  MoveL 11373 to (499.02, 502.81, 19.8) mm, rotated rx 0 ry 90 rz 0 deg; joints [-12.285, -28.387, 111.814, -16.313, -82.826, 51.071]
  Set speed (15.0 mm/s)
  Call Extruder(0.024)
  MoveL 11374 to (498.43, 503.4, 19.8) mm, rotated rx 0 ry 90 rz 0 deg; joints [-12.351, -28.396, 111.869, -16.378, -82.873, 51.065]
  Set speed (120.0 mm/s)
  MoveL 11375 to (496.44, 504.19, 19.8) mm, rotated rx 0 ry 90 rz 0 deg; joints [-12.464, -28.43, 112.084, -16.485, -83.05, 51.026]
  Set speed (1000.0 mm/s)
  MoveL 11376 to (495, 504.85, 19.8) mm, rotated rx 0 ry 90 rz 0 deg; joints [-12.554, -28.454, 112.239, -16.571, -83.178, 50.998]
  Set speed (15.0 mm/s)
  Call Extruder(0.148)
  MoveL 11377 to (491.4, 508.44, 19.8) mm, rotated rx 0 ry 90 rz 0 deg; joints [-12.96, -28.505, 112.569, -16.971, -83.458, 50.958]
  Set speed (120.0 mm/s)
  MoveL 11378 to (492.24, 508.59, 19.8) mm, rotated rx 0 ry 90 rz 0 deg; joints [-12.956, -28.489, 112.465, -16.97, -83.374, 50.983]
  Set speed (15.0 mm/s)
  Call Extruder(0.113)
  MoveL 11379 to (495, 505.84, 19.8) mm, rotated rx 0 ry 90 rz 0 deg; joints [-12.645, -28.45, 112.212, -16.664, -83.16, 51.014]
  Set speed (120.0 mm/s)
  MoveL 11380 to (495, 506.83, 19.8) mm, rotated rx 0 ry 90 rz 0 deg; joints [-12.735, -28.446, 112.186, -16.756, -83.141, 51.03]
  Set speed (15.0 mm/s)
  Call Extruder(0.073)
  MoveL 11381 to (493.23, 508.59, 19.8) mm, rotated rx 0 ry 90 rz 0 deg; joints [-12.935, -28.471, 112.348, -16.952, -83.278, 51.01]
  Set speed (120.0 mm/s)
  MoveL 11382 to (494.22, 508.59, 19.8) mm, rotated rx 0 ry 90 rz 0 deg; joints [-12.914, -28.453, 112.23, -16.934, -83.183, 51.037]
  Set speed (15.0 mm/s)
  Call Extruder(0.036)
  MoveL 11383 to (495.1, 507.72, 19.8) mm, rotated rx 0 ry 90 rz 0 deg; joints [-12.816, -28.441, 112.15, -16.838, -83.115, 51.047]
  Set speed (120.0 mm/s)
  MoveL 11384 to (495.21, 508.59, 19.8) mm, rotated rx 0 ry 90 rz 0 deg; joints [-12.893, -28.435, 112.113, -16.917, -83.087, 51.064]
  Set speed (15.0 mm/s)
  MoveL 11385 to (496.09, 507.72, 19.8) mm, rotated rx 0 ry 90 rz 0 deg; joints [-12.795, -28.422, 112.033, -16.82, -83.019, 51.074]
  Set speed (120.0 mm/s)
  MoveL 11386 to (496.2, 508.59, 19.8) mm, rotated rx 0 ry 90 rz 0 deg; joints [-12.872, -28.416, 111.995, -16.899, -82.992, 51.091]
  Set speed (15.0 mm/s)
  Call Extruder(0.036)
  MoveL 11387 to (497.08, 507.72, 19.8) mm, rotated rx 0 ry 90 rz 0 deg; joints [-12.774, -28.403, 111.915, -16.803, -82.924, 51.1]
  Set speed (120.0 mm/s)
  MoveL 11388 to (497.19, 508.59, 19.8) mm, rotated rx 0 ry 90 rz 0 deg; joints [-12.852, -28.397, 111.877, -16.882, -82.896, 51.118]
  Set speed (15.0 mm/s)
  MoveL 11389 to (498.07, 507.72, 19.8) mm, rotated rx 0 ry 90 rz 0 deg; joints [-12.754, -28.385, 111.797, -16.786, -82.828, 51.127]
  Set speed (120.0 mm/s)
  MoveL 11390 to (498.18, 508.59, 19.8) mm, rotated rx 0 ry 90 rz 0 deg; joints [-12.831, -28.379, 111.759, -16.865, -82.801, 51.145]
  Set speed (15.0 mm/s)
  MoveL 11391 to (499.06, 507.72, 19.8) mm, rotated rx 0 ry 90 rz 0 deg; joints [-12.733, -28.366, 111.679, -16.769, -82.733, 51.153]
  Set speed (120.0 mm/s)
  MoveL 11392 to (499.17, 508.59, 19.8) mm, rotated rx 0 ry 90 rz 0 deg; joints [-12.811, -28.36, 111.641, -16.848, -82.705, 51.171]
  Set speed (15.0 mm/s)
  MoveL 11393 to (500.05, 507.72, 19.8) mm, rotated rx 0 ry 90 rz 0 deg; joints [-12.713, -28.347, 111.561, -16.752, -82.637, 51.18]
  Set speed (120.0 mm/s)
  MoveL 11394 to (500.16, 508.59, 19.8) mm, rotated rx 0 ry 90 rz 0 deg; joints [-12.79, -28.34, 111.523, -16.831, -82.61, 51.198]
  Set speed (15.0 mm/s)
  MoveL 11395 to (501.04, 507.72, 19.8) mm, rotated rx 0 ry 90 rz 0 deg; joints [-12.693, -28.327, 111.443, -16.735, -82.542, 51.206]
  Set speed (120.0 mm/s)
  MoveL 11396 to (501.15, 508.59, 19.8) mm, rotated rx 0 ry 90 rz 0 deg; joints [-12.77, -28.321, 111.405, -16.814, -82.514, 51.224]
  Set speed (15.0 mm/s)
  MoveL 11397 to (502.03, 507.72, 19.8) mm, rotated rx 0 ry 90 rz 0 deg; joints [-12.672, -28.308, 111.324, -16.719, -82.446, 51.233]
  Set speed (120.0 mm/s)
  MoveL 11398 to (502.14, 508.59, 19.8) mm, rotated rx 0 ry 90 rz 0 deg; joints [-12.749, -28.302, 111.287, -16.797, -82.419, 51.251]
  Set speed (15.0 mm/s)
  MoveL 11399 to (503.02, 507.72, 19.8) mm, rotated rx 0 ry 90 rz 0 deg; joints [-12.652, -28.288, 111.206, -16.702, -82.351, 51.259]
  Set speed (120.0 mm/s)
  MoveL 11400 to (503.13, 508.59, 19.8) mm, rotated rx 0 ry 90 rz 0 deg; joints [-12.729, -28.282, 111.168, -16.781, -82.324, 51.277]
  Set speed (15.0 mm/s)
  MoveL 11401 to (504.01, 507.72, 19.8) mm, rotated rx 0 ry 90 rz 0 deg; joints [-12.632, -28.268, 111.087, -16.686, -82.255, 51.285]
  Set speed (120.0 mm/s)
  MoveL 11402 to (504.12, 508.59, 19.8) mm, rotated rx 0 ry 90 rz 0 deg; joints [-12.709, -28.262, 111.049, -16.764, -82.228, 51.304]
  Set speed (15.0 mm/s)
  MoveL 11403 to (505, 507.72, 19.8) mm, rotated rx 0 ry 90 rz 0 deg; joints [-12.612, -28.249, 110.968, -16.669, -82.16, 51.311]
  Set speed (120.0 mm/s)
  MoveL 11404 to (505.33, 507.39, 19.8) mm, rotated rx 0 ry 90 rz 0 deg; joints [-12.575, -28.243, 110.937, -16.633, -82.134, 51.314]
  Set speed (15.0 mm/s)
  Call Extruder(0.134)
  MoveL 11405 to (508.59, 504.12, 19.8) mm, rotated rx 0 ry 90 rz 0 deg; joints [-12.216, -28.191, 110.631, -16.281, -81.877, 51.342]
  Set speed (120.0 mm/s)
  MoveL 11406 to (508.59, 505.11, 19.8) mm, rotated rx 0 ry 90 rz 0 deg; joints [-12.305, -28.187, 110.605, -16.371, -81.86, 51.36]
  Set speed (15.0 mm/s)
  Call Extruder(0.143)
  MoveL 11407 to (505.11, 508.59, 19.8) mm, rotated rx 0 ry 90 rz 0 deg; joints [-12.689, -28.242, 110.931, -16.748, -82.133, 51.33]
  Set speed (120.0 mm/s)
  MoveL 11408 to (506.1, 508.59, 19.8) mm, rotated rx 0 ry 90 rz 0 deg; joints [-12.668, -28.222, 110.812, -16.732, -82.038, 51.356]
  Set speed (15.0 mm/s)
  Call Extruder(0.103)
  MoveL 11409 to (508.59, 506.1, 19.8) mm, rotated rx 0 ry 90 rz 0 deg; joints [-12.394, -28.182, 110.579, -16.462, -81.842, 51.377]
  Set speed (120.0 mm/s)
  MoveL 11410 to (508.59, 507.09, 19.8) mm, rotated rx 0 ry 90 rz 0 deg; joints [-12.483, -28.178, 110.552, -16.553, -81.825, 51.395]
  Set speed (15.0 mm/s)
  Call Extruder(0.062)
  MoveL 11411 to (507.09, 508.59, 19.8) mm, rotated rx 0 ry 90 rz 0 deg; joints [-12.648, -28.202, 110.693, -16.715, -81.942, 51.382]
  Set speed (120.0 mm/s)
  MoveL 11412 to (508.08, 508.59, 19.8) mm, rotated rx 0 ry 90 rz 0 deg; joints [-12.628, -28.181, 110.574, -16.699, -81.847, 51.408]
  Set speed (15.0 mm/s)
  Call Extruder(0.021)
  MoveL 11413 to (508.59, 508.08, 19.8) mm, rotated rx 0 ry 90 rz 0 deg; joints [-12.572, -28.173, 110.526, -16.644, -81.807, 51.413]
  Set speed (120.0 mm/s)
  MoveL 11414 to (505.33, 506.39, 19.8) mm, rotated rx 0 ry 90 rz 0 deg; joints [-12.485, -28.248, 110.963, -16.542, -82.152, 51.297]
  Set speed (15.0 mm/s)
  Call Extruder(0.134)
  MoveL 11415 to (508.59, 503.13, 19.8) mm, rotated rx 0 ry 90 rz 0 deg; joints [-12.126, -28.195, 110.656, -16.19, -81.894, 51.325]
  Set speed (120.0 mm/s)
  MoveL 11416 to (508.59, 502.14, 19.8) mm, rotated rx 0 ry 90 rz 0 deg; joints [-12.037, -28.2, 110.682, -16.099, -81.911, 51.307]
  Set speed (15.0 mm/s)
  Call Extruder(0.136)
  MoveL 11417 to (505.28, 505.46, 19.8) mm, rotated rx 0 ry 90 rz 0 deg; joints [-12.402, -28.253, 110.994, -16.456, -82.173, 51.279]
  Set speed (120.0 mm/s)
  MoveL 11418 to (504.94, 504.8, 19.8) mm, rotated rx 0 ry 90 rz 0 deg; joints [-12.349, -28.263, 111.052, -16.401, -82.217, 51.259]
  Set speed (15.0 mm/s)
  Call Extruder(0.150)
  MoveL 11419 to (508.59, 501.15, 19.8) mm, rotated rx 0 ry 90 rz 0 deg; joints [-11.948, -28.204, 110.707, -16.008, -81.928, 51.29]
  Set speed (120.0 mm/s)
  MoveL 11420 to (508.59, 500.16, 19.8) mm, rotated rx 0 ry 90 rz 0 deg; joints [-11.858, -28.208, 110.732, -15.916, -81.945, 51.273]
  Set speed (15.0 mm/s)
  Call Extruder(0.164)
  MoveL 11421 to (504.61, 504.15, 19.8) mm, rotated rx 0 ry 90 rz 0 deg; joints [-12.296, -28.272, 111.109, -16.346, -82.261, 51.239]
  Set speed (120.0 mm/s)
  MoveL 11422 to (504.27, 503.49, 19.8) mm, rotated rx 0 ry 90 rz 0 deg; joints [-12.243, -28.282, 111.167, -16.291, -82.305, 51.219]
  Set speed (15.0 mm/s)
  Call Extruder(0.178)
  MoveL 11423 to (508.59, 499.17, 19.8) mm, rotated rx 0 ry 90 rz 0 deg; joints [-11.769, -28.213, 110.757, -15.825, -81.962, 51.256]
  Set speed (120.0 mm/s)
  MoveL 11424 to (508.59, 498.18, 19.8) mm, rotated rx 0 ry 90 rz 0 deg; joints [-11.679, -28.217, 110.782, -15.734, -81.978, 51.239]
  Set speed (15.0 mm/s)
  Call Extruder(0.192)
  MoveL 11425 to (503.94, 502.84, 19.8) mm, rotated rx 0 ry 90 rz 0 deg; joints [-12.191, -28.291, 111.224, -16.236, -82.349, 51.2]
  Set speed (120.0 mm/s)
  MoveL 11426 to (503.6, 502.18, 19.8) mm, rotated rx 0 ry 90 rz 0 deg; joints [-12.138, -28.301, 111.281, -16.181, -82.393, 51.18]
  Set speed (15.0 mm/s)
  Call Extruder(0.205)
  MoveL 11427 to (508.59, 497.19, 19.8) mm, rotated rx 0 ry 90 rz 0 deg; joints [-11.589, -28.221, 110.807, -15.643, -81.995, 51.222]
  Set speed (120.0 mm/s)
  MoveL 11428 to (508.59, 496.2, 19.8) mm, rotated rx 0 ry 90 rz 0 deg; joints [-11.5, -28.225, 110.831, -15.552, -82.011, 51.206]
  Set speed (15.0 mm/s)
  Call Extruder(0.219)
  MoveL 11429 to (503.27, 501.53, 19.8) mm, rotated rx 0 ry 90 rz 0 deg; joints [-12.084, -28.31, 111.338, -16.126, -82.437, 51.16]
  Set speed (120.0 mm/s)
  MoveL 11430 to (502.93, 500.87, 19.8) mm, rotated rx 0 ry 90 rz 0 deg; joints [-12.031, -28.32, 111.395, -16.07, -82.481, 51.141]
  Set speed (15.0 mm/s)
  Call Extruder(0.233)
  MoveL 11431 to (508.59, 495.21, 19.8) mm, rotated rx 0 ry 90 rz 0 deg; joints [-11.41, -28.229, 110.855, -15.46, -82.028, 51.189]
  Set speed (120.0 mm/s)
  MoveL 11432 to (508.59, 494.22, 19.8) mm, rotated rx 0 ry 90 rz 0 deg; joints [-11.32, -28.234, 110.879, -15.369, -82.044, 51.172]
  Set speed (15.0 mm/s)
  Call Extruder(0.247)
  MoveL 11433 to (502.6, 500.22, 19.8) mm, rotated rx 0 ry 90 rz 0 deg; joints [-11.978, -28.329, 111.452, -16.015, -82.525, 51.121]
  Set speed (120.0 mm/s)
  MoveL 11434 to (502.26, 499.57, 19.8) mm, rotated rx 0 ry 90 rz 0 deg; joints [-11.925, -28.338, 111.509, -15.96, -82.569, 51.102]
  Set speed (15.0 mm/s)
  Call Extruder(0.109)
  MoveL 11435 to (504.9, 496.92, 19.8) mm, rotated rx 0 ry 90 rz 0 deg; joints [-11.634, -28.297, 111.258, -15.674, -82.358, 51.125]
  Set speed (120.0 mm/s)
  MoveL 11436 to (505.52, 496.31, 19.8) mm, rotated rx 0 ry 90 rz 0 deg; joints [-11.567, -28.287, 111.199, -15.608, -82.309, 51.131]
  Set speed (15.0 mm/s)
  Call Extruder(0.127)
  MoveL 11437 to (508.59, 493.23, 19.8) mm, rotated rx 0 ry 90 rz 0 deg; joints [-11.23, -28.238, 110.903, -15.277, -82.06, 51.156]
  Set speed (120.0 mm/s)
  MoveL 11438 to (508.59, 492.24, 19.8) mm, rotated rx 0 ry 90 rz 0 deg; joints [-11.14, -28.242, 110.927, -15.186, -82.076, 51.139]
  Set speed (15.0 mm/s)
  MoveL 11439 to (505.52, 495.32, 19.8) mm, rotated rx 0 ry 90 rz 0 deg; joints [-11.476, -28.291, 111.224, -15.516, -82.325, 51.114]
  Set speed (120.0 mm/s)
  MoveL 11440 to (505.52, 494.33, 19.8) mm, rotated rx 0 ry 90 rz 0 deg; joints [-11.386, -28.295, 111.248, -15.424, -82.342, 51.098]
  Set speed (15.0 mm/s)
  Call Extruder(0.121)
  MoveL 11441 to (508.44, 491.4, 19.8) mm, rotated rx 0 ry 90 rz 0 deg; joints [-11.067, -28.248, 110.965, -15.11, -82.104, 51.122]
  Set speed (120.0 mm/s)
  MoveL 11442 to (507.45, 491.4, 19.8) mm, rotated rx 0 ry 90 rz 0 deg; joints [-11.084, -28.268, 111.084, -15.125, -82.2, 51.098]
  Set speed (15.0 mm/s)
  Call Extruder(0.080)
  MoveL 11443 to (505.52, 493.34, 19.8) mm, rotated rx 0 ry 90 rz 0 deg; joints [-11.296, -28.299, 111.272, -15.333, -82.358, 51.082]
  Set speed (120.0 mm/s)
  MoveL 11444 to (505.27, 492.6, 19.8) mm, rotated rx 0 ry 90 rz 0 deg; joints [-11.233, -28.307, 111.32, -15.268, -82.394, 51.064]
  Set speed (15.0 mm/s)
  Call Extruder(0.049)
  MoveL 11445 to (506.46, 491.4, 19.8) mm, rotated rx 0 ry 90 rz 0 deg; joints [-11.102, -28.288, 111.204, -15.139, -82.297, 51.074]
  Set speed (120.0 mm/s)
  MoveL 11446 to (505.47, 491.4, 19.8) mm, rotated rx 0 ry 90 rz 0 deg; joints [-11.12, -28.308, 111.323, -15.153, -82.393, 51.05]
  Set speed (15.0 mm/s)
  MoveL 11447 to (504.28, 492.6, 19.8) mm, rotated rx 0 ry 90 rz 0 deg; joints [-11.251, -28.327, 111.439, -15.282, -82.491, 51.04]
  Set speed (120.0 mm/s)
  MoveL 11448 to (503.29, 492.6, 19.8) mm, rotated rx 0 ry 90 rz 0 deg; joints [-11.269, -28.346, 111.558, -15.297, -82.587, 51.015]
  Set speed (15.0 mm/s)
  MoveL 11449 to (504.48, 491.4, 19.8) mm, rotated rx 0 ry 90 rz 0 deg; joints [-11.137, -28.327, 111.442, -15.168, -82.49, 51.026]
  Set speed (120.0 mm/s)
  MoveL 11450 to (503.49, 491.4, 19.8) mm, rotated rx 0 ry 90 rz 0 deg; joints [-11.155, -28.347, 111.561, -15.182, -82.587, 51.001]
  Set speed (15.0 mm/s)
  MoveL 11451 to (502.3, 492.6, 19.8) mm, rotated rx 0 ry 90 rz 0 deg; joints [-11.287, -28.365, 111.676, -15.312, -82.684, 50.991]
  Set speed (120.0 mm/s)
  MoveL 11452 to (501.31, 492.6, 19.8) mm, rotated rx 0 ry 90 rz 0 deg; joints [-11.305, -28.384, 111.795, -15.327, -82.781, 50.966]
  Set speed (15.0 mm/s)
  MoveL 11453 to (502.5, 491.4, 19.8) mm, rotated rx 0 ry 90 rz 0 deg; joints [-11.173, -28.366, 111.68, -15.197, -82.683, 50.977]
  Set speed (120.0 mm/s)
  MoveL 11454 to (501.51, 491.4, 19.8) mm, rotated rx 0 ry 90 rz 0 deg; joints [-11.191, -28.385, 111.799, -15.212, -82.78, 50.953]
  Set speed (15.0 mm/s)
  MoveL 11455 to (500.32, 492.6, 19.8) mm, rotated rx 0 ry 90 rz 0 deg; joints [-11.323, -28.403, 111.914, -15.342, -82.877, 50.942]
  Set speed (120.0 mm/s)
  MoveL 11456 to (499.33, 492.6, 19.8) mm, rotated rx 0 ry 90 rz 0 deg; joints [-11.342, -28.422, 112.032, -15.357, -82.974, 50.917]
  Set speed (15.0 mm/s)
  MoveL 11457 to (500.52, 491.4, 19.8) mm, rotated rx 0 ry 90 rz 0 deg; joints [-11.209, -28.404, 111.917, -15.227, -82.877, 50.928]
  Set speed (120.0 mm/s)
  MoveL 11458 to (499.53, 491.4, 19.8) mm, rotated rx 0 ry 90 rz 0 deg; joints [-11.227, -28.423, 112.036, -15.242, -82.974, 50.904]
  Set speed (15.0 mm/s)
  Call Extruder(0.049)
  MoveL 11459 to (498.34, 492.6, 19.8) mm, rotated rx 0 ry 90 rz 0 deg; joints [-11.36, -28.441, 112.15, -15.372, -83.071, 50.893]
  Set speed (120.0 mm/s)
  MoveL 11460 to (497.35, 492.6, 19.8) mm, rotated rx 0 ry 90 rz 0 deg; joints [-11.378, -28.459, 112.268, -15.387, -83.167, 50.868]
  Set speed (15.0 mm/s)
  MoveL 11461 to (498.54, 491.4, 19.8) mm, rotated rx 0 ry 90 rz 0 deg; joints [-11.245, -28.441, 112.154, -15.257, -83.07, 50.88]
  Set speed (120.0 mm/s)
  MoveL 11462 to (497.55, 491.4, 19.8) mm, rotated rx 0 ry 90 rz 0 deg; joints [-11.264, -28.46, 112.272, -15.272, -83.167, 50.855]
  Set speed (15.0 mm/s)
  MoveL 11463 to (496.36, 492.6, 19.8) mm, rotated rx 0 ry 90 rz 0 deg; joints [-11.397, -28.477, 112.386, -15.403, -83.264, 50.843]
  MoveL 11464 to (496.23, 492.73, 19.8) mm, rotated rx 0 ry 90 rz 0 deg; joints [-11.41, -28.479, 112.398, -15.416, -83.274, 50.842]
  Set speed (120.0 mm/s)
  MoveL 11465 to (504.54, 493.58, 19.8) mm, rotated rx 0 ry 90 rz 0 deg; joints [-11.335, -28.318, 111.383, -15.369, -82.449, 51.062]
  Set speed (1000.0 mm/s)
  MoveL 11466 to (504.54, 495.95, 19.8) mm, rotated rx 0 ry 90 rz 0 deg; joints [-11.552, -28.308, 111.326, -15.589, -82.41, 51.1]
  Set speed (1000.0 mm/s)
  MoveL 11467 to (501.26, 497.6, 19.8) mm, rotated rx 0 ry 90 rz 0 deg; joints [-11.764, -28.366, 111.679, -15.793, -82.701, 51.044]
  Set speed (15.0 mm/s)
  Call Extruder(0.028)
  MoveL 11468 to (501.93, 496.92, 19.8) mm, rotated rx 0 ry 90 rz 0 deg; joints [-11.69, -28.355, 111.614, -15.719, -82.647, 51.051]
  Set speed (120.0 mm/s)
  MoveL 11469 to (502.92, 496.92, 19.8) mm, rotated rx 0 ry 90 rz 0 deg; joints [-11.671, -28.336, 111.496, -15.704, -82.55, 51.076]
  Set speed (15.0 mm/s)
  Call Extruder(0.055)
  MoveL 11470 to (501.59, 498.26, 19.8) mm, rotated rx 0 ry 90 rz 0 deg; joints [-11.818, -28.357, 111.622, -15.849, -82.657, 51.063]
  Set speed (120.0 mm/s)
  MoveL 11471 to (501.93, 498.91, 19.8) mm, rotated rx 0 ry 90 rz 0 deg; joints [-11.871, -28.347, 111.565, -15.904, -82.613, 51.083]
  Set speed (15.0 mm/s)
  Call Extruder(0.082)
  MoveL 11472 to (503.91, 496.92, 19.8) mm, rotated rx 0 ry 90 rz 0 deg; joints [-11.652, -28.317, 111.377, -15.689, -82.454, 51.101]
  MoveL 11473 to (504.04, 496.8, 19.8) mm, rotated rx 0 ry 90 rz 0 deg; joints [-11.639, -28.315, 111.365, -15.676, -82.444, 51.102]
  Set speed (120.0 mm/s)
  MoveL 11474 to (504.37, 505.79, 19.8) mm, rotated rx 0 ry 90 rz 0 deg; joints [-12.45, -28.27, 111.095, -16.502, -82.256, 51.261]
  Set speed (1000.0 mm/s)
  MoveL 11475 to (490.47, 509.53, 19.8) mm, rotated rx 0 ry 90 rz 0 deg; joints [-13.08, -28.517, 112.649, -17.089, -83.527, 50.95]
  Set speed (1000.0 mm/s)
  MoveL 11476 to (490.4, 509.6, 19.8) mm, rotated rx 0 ry 90 rz 0 deg; joints [-13.088, -28.518, 112.656, -17.097, -83.532, 50.949]
  Set speed (1000.0 mm/s)
  MoveL 11477 to (490.4, 509.6, 19.9) mm, rotated rx 0 ry 90 rz 0 deg; joints [-13.088, -28.529, 112.661, -17.097, -83.527, 50.951]
  Set speed (15.0 mm/s)
  Call Extruder(0.559)
  MoveL 11478 to (490.4, 490.4, 19.9) mm, rotated rx 0 ry 90 rz 0 deg; joints [-11.303, -28.602, 113.152, -15.29, -83.88, 50.663]
  MoveL 11479 to (509.6, 490.4, 19.9) mm, rotated rx 0 ry 90 rz 0 deg; joints [-10.955, -28.239, 110.854, -15.001, -82.002, 51.135]
  MoveL 11480 to (509.6, 509.6, 19.9) mm, rotated rx 0 ry 90 rz 0 deg; joints [-12.688, -28.155, 110.368, -16.767, -81.678, 51.468]
  MoveL 11481 to (490.4, 509.6, 19.9) mm, rotated rx 0 ry 90 rz 0 deg; joints [-13.088, -28.529, 112.661, -17.097, -83.527, 50.951]
  Set speed (120.0 mm/s)
  MoveL 11482 to (490.4, 509.2, 19.9) mm, rotated rx 0 ry 90 rz 0 deg; joints [-13.051, -28.53, 112.672, -17.06, -83.535, 50.944]
  Set speed (1000.0 mm/s)
  MoveL 11483 to (490.5, 509.2, 19.9) mm, rotated rx 0 ry 90 rz 0 deg; joints [-13.049, -28.529, 112.66, -17.058, -83.525, 50.947]
  Set speed (1000.0 mm/s)
  MoveL 11484 to (495.94, 504.34, 19.9) mm, rotated rx 0 ry 90 rz 0 deg; joints [-12.487, -28.45, 112.146, -16.508, -83.092, 51.016]
  Set speed (1000.0 mm/s)
  MoveL 11485 to (496.01, 504.4, 19.9) mm, rotated rx 0 ry 90 rz 0 deg; joints [-12.492, -28.448, 112.136, -16.513, -83.084, 51.019]
  Set speed (15.0 mm/s)
  Call Extruder(0.067)
  MoveL 11486 to (496.01, 506.72, 19.9) mm, rotated rx 0 ry 90 rz 0 deg; joints [-12.705, -28.438, 112.074, -16.728, -83.041, 51.057]
  Call Extruder(0.242)
  MoveL 11487 to (504.33, 506.72, 19.9) mm, rotated rx 0 ry 90 rz 0 deg; joints [-12.535, -28.277, 111.08, -16.588, -82.237, 51.278]
  Call Extruder(0.027)
  MoveL 11488 to (504.33, 505.8, 19.9) mm, rotated rx 0 ry 90 rz 0 deg; joints [-12.452, -28.281, 111.105, -16.504, -82.254, 51.262]
  Call Extruder(0.306)
  MoveL 11489 to (499.53, 496.43, 19.9) mm, rotated rx 0 ry 90 rz 0 deg; joints [-11.69, -28.414, 111.919, -15.711, -82.884, 50.983]
  Call Extruder(0.017)
  MoveL 11490 to (499.27, 495.92, 19.9) mm, rotated rx 0 ry 90 rz 0 deg; joints [-11.648, -28.421, 111.963, -15.668, -82.918, 50.969]
  Call Extruder(0.010)
  MoveL 11491 to (499.84, 495.92, 19.9) mm, rotated rx 0 ry 90 rz 0 deg; joints [-11.637, -28.41, 111.895, -15.659, -82.862, 50.983]
  Call Extruder(0.000)
  MoveL 11492 to (499.84, 495.92, 19.9) mm, rotated rx 0 ry 90 rz 0 deg; joints [-11.637, -28.41, 111.895, -15.659, -82.862, 50.983]
  Call Extruder(0.136)
  MoveL 11493 to (504.51, 495.92, 19.9) mm, rotated rx 0 ry 90 rz 0 deg; joints [-11.55, -28.319, 111.335, -15.587, -82.408, 51.101]
  Call Extruder(0.067)
  MoveL 11494 to (504.51, 493.61, 19.9) mm, rotated rx 0 ry 90 rz 0 deg; joints [-11.338, -28.329, 111.391, -15.372, -82.446, 51.063]
  Call Extruder(0.250)
  MoveL 11495 to (495.92, 493.61, 19.9) mm, rotated rx 0 ry 90 rz 0 deg; joints [-11.498, -28.492, 112.419, -15.504, -83.284, 50.849]
  Call Extruder(0.027)
  MoveL 11496 to (495.92, 494.52, 19.9) mm, rotated rx 0 ry 90 rz 0 deg; joints [-11.583, -28.489, 112.397, -15.59, -83.268, 50.863]
  Call Extruder(0.306)
  MoveL 11497 to (500.7, 503.9, 19.9) mm, rotated rx 0 ry 90 rz 0 deg; joints [-12.351, -28.361, 111.589, -16.387, -82.638, 51.135]
  Call Extruder(0.017)
  MoveL 11498 to (500.96, 504.4, 19.9) mm, rotated rx 0 ry 90 rz 0 deg; joints [-12.392, -28.354, 111.545, -16.43, -82.604, 51.15]
  Call Extruder(0.010)
  MoveL 11499 to (500.39, 504.41, 19.9) mm, rotated rx 0 ry 90 rz 0 deg; joints [-12.404, -28.365, 111.613, -16.439, -82.659, 51.135]
  Call Extruder(0.000)
  MoveL 11500 to (500.39, 504.41, 19.9) mm, rotated rx 0 ry 90 rz 0 deg; joints [-12.404, -28.365, 111.613, -16.439, -82.659, 51.135]
  Call Extruder(0.128)
  MoveL 11501 to (496.01, 504.4, 19.9) mm, rotated rx 0 ry 90 rz 0 deg; joints [-12.492, -28.448, 112.136, -16.513, -83.084, 51.019]
  Set speed (120.0 mm/s)
  MoveL 11502 to (496.01, 504.81, 19.9) mm, rotated rx 0 ry 90 rz 0 deg; joints [-12.529, -28.446, 112.125, -16.55, -83.076, 51.025]
  Set speed (1000.0 mm/s)
  MoveL 11503 to (495.91, 504.81, 19.9) mm, rotated rx 0 ry 90 rz 0 deg; joints [-12.531, -28.448, 112.137, -16.552, -83.086, 51.023]
  Set speed (1000.0 mm/s)
  MoveL 11504 to (495.32, 503.72, 19.9) mm, rotated rx 0 ry 90 rz 0 deg; joints [-12.443, -28.464, 112.236, -16.46, -83.163, 50.99]
  Set speed (15.0 mm/s)
  Call Extruder(0.107)
  MoveL 11505 to (495.32, 507.41, 19.9) mm, rotated rx 0 ry 90 rz 0 deg; joints [-12.782, -28.448, 112.138, -16.805, -83.094, 51.049]
  Call Extruder(0.282)
  MoveL 11506 to (505.02, 507.41, 19.9) mm, rotated rx 0 ry 90 rz 0 deg; joints [-12.583, -28.26, 110.979, -16.64, -82.158, 51.308]
  Call Extruder(0.052)
  MoveL 11507 to (505.02, 505.64, 19.9) mm, rotated rx 0 ry 90 rz 0 deg; joints [-12.423, -28.268, 111.026, -16.477, -82.19, 51.277]
  Call Extruder(0.295)
  MoveL 11508 to (500.4, 496.61, 19.9) mm, rotated rx 0 ry 90 rz 0 deg; joints [-11.69, -28.397, 111.811, -15.714, -82.796, 51.008]
  Call Extruder(0.140)
  MoveL 11509 to (505.2, 496.61, 19.9) mm, rotated rx 0 ry 90 rz 0 deg; joints [-11.6, -28.303, 111.235, -15.64, -82.329, 51.129]
  Call Extruder(0.107)
  MoveL 11510 to (505.2, 492.92, 19.9) mm, rotated rx 0 ry 90 rz 0 deg; joints [-11.263, -28.318, 111.325, -15.298, -82.39, 51.069]
  Call Extruder(0.290)
  MoveL 11511 to (495.23, 492.92, 19.9) mm, rotated rx 0 ry 90 rz 0 deg; joints [-11.447, -28.507, 112.518, -15.45, -83.363, 50.821]
  Call Extruder(0.052)
  MoveL 11512 to (495.23, 494.69, 19.9) mm, rotated rx 0 ry 90 rz 0 deg; joints [-11.611, -28.501, 112.475, -15.617, -83.333, 50.848]
  Call Extruder(0.295)
  MoveL 11513 to (499.84, 503.72, 19.9) mm, rotated rx 0 ry 90 rz 0 deg; joints [-12.352, -28.378, 111.697, -16.384, -82.726, 51.109]
  Call Extruder(0.132)
  MoveL 11514 to (495.32, 503.72, 19.9) mm, rotated rx 0 ry 90 rz 0 deg; joints [-12.443, -28.464, 112.236, -16.46, -83.163, 50.99]
  Set speed (120.0 mm/s)
  MoveL 11515 to (491.09, 508.91, 19.9) mm, rotated rx 0 ry 90 rz 0 deg; joints [-13.01, -28.519, 112.598, -17.02, -83.474, 50.959]
  Set speed (15.0 mm/s)
  Call Extruder(0.519)
  MoveL 11516 to (491.09, 491.09, 19.9) mm, rotated rx 0 ry 90 rz 0 deg; joints [-11.355, -28.587, 113.054, -15.344, -83.8, 50.69]
  MoveL 11517 to (508.91, 491.09, 19.9) mm, rotated rx 0 ry 90 rz 0 deg; joints [-11.03, -28.25, 110.921, -15.075, -82.058, 51.13]
  MoveL 11518 to (508.91, 508.91, 19.9) mm, rotated rx 0 ry 90 rz 0 deg; joints [-12.64, -28.173, 110.47, -16.715, -81.757, 51.437]
  MoveL 11519 to (491.09, 508.91, 19.9) mm, rotated rx 0 ry 90 rz 0 deg; joints [-13.01, -28.519, 112.598, -17.02, -83.474, 50.959]
  Set speed (120.0 mm/s)
  MoveL 11520 to (491.76, 508.59, 19.9) mm, rotated rx 0 ry 90 rz 0 deg; joints [-12.966, -28.508, 112.527, -16.978, -83.415, 50.972]
  Set speed (15.0 mm/s)
  Call Extruder(0.015)
  MoveL 11521 to (491.4, 508.23, 19.9) mm, rotated rx 0 ry 90 rz 0 deg; joints [-12.94, -28.516, 112.579, -16.951, -83.457, 50.956]
  Set speed (120.0 mm/s)
  MoveL 11522 to (491.4, 507.24, 19.9) mm, rotated rx 0 ry 90 rz 0 deg; joints [-12.849, -28.521, 112.606, -16.858, -83.476, 50.941]
  Set speed (15.0 mm/s)
  Call Extruder(0.056)
  MoveL 11523 to (492.75, 508.59, 19.9) mm, rotated rx 0 ry 90 rz 0 deg; joints [-12.945, -28.491, 112.41, -16.961, -83.319, 50.999]
  Set speed (120.0 mm/s)
  MoveL 11524 to (493.74, 508.59, 19.9) mm, rotated rx 0 ry 90 rz 0 deg; joints [-12.924, -28.472, 112.292, -16.943, -83.224, 51.026]
  Set speed (15.0 mm/s)
  Call Extruder(0.096)
  MoveL 11525 to (491.4, 506.25, 19.9) mm, rotated rx 0 ry 90 rz 0 deg; joints [-12.758, -28.525, 112.633, -16.766, -83.495, 50.925]
  Set speed (120.0 mm/s)
  MoveL 11526 to (491.4, 505.26, 19.9) mm, rotated rx 0 ry 90 rz 0 deg; joints [-12.666, -28.529, 112.659, -16.673, -83.513, 50.909]
  Set speed (15.0 mm/s)
  Call Extruder(0.137)
  MoveL 11527 to (494.74, 508.59, 19.9) mm, rotated rx 0 ry 90 rz 0 deg; joints [-12.903, -28.454, 112.175, -16.925, -83.128, 51.053]
  Set speed (120.0 mm/s)
  MoveL 11528 to (495.72, 508.59, 19.9) mm, rotated rx 0 ry 90 rz 0 deg; joints [-12.882, -28.436, 112.057, -16.908, -83.033, 51.08]
  Set speed (15.0 mm/s)
  Call Extruder(0.178)
  MoveL 11529 to (491.4, 504.27, 19.9) mm, rotated rx 0 ry 90 rz 0 deg; joints [-12.574, -28.533, 112.685, -16.58, -83.532, 50.894]
  Set speed (120.0 mm/s)
  MoveL 11530 to (491.4, 503.28, 19.9) mm, rotated rx 0 ry 90 rz 0 deg; joints [-12.483, -28.536, 112.711, -16.487, -83.551, 50.879]
  Set speed (15.0 mm/s)
  Call Extruder(0.148)
  MoveL 11531 to (495, 506.88, 19.9) mm, rotated rx 0 ry 90 rz 0 deg; joints [-12.74, -28.456, 112.189, -16.761, -83.135, 51.032]
  Set speed (120.0 mm/s)
  MoveL 11532 to (495, 505.89, 19.9) mm, rotated rx 0 ry 90 rz 0 deg; joints [-12.649, -28.461, 112.216, -16.669, -83.153, 51.016]
  Set speed (15.0 mm/s)
  Call Extruder(0.148)
  MoveL 11533 to (491.4, 502.29, 19.9) mm, rotated rx 0 ry 90 rz 0 deg; joints [-12.391, -28.54, 112.737, -16.394, -83.569, 50.863]
  Set speed (120.0 mm/s)
  MoveL 11534 to (491.4, 501.3, 19.9) mm, rotated rx 0 ry 90 rz 0 deg; joints [-12.299, -28.544, 112.763, -16.301, -83.587, 50.848]
  Set speed (15.0 mm/s)
  MoveL 11535 to (495, 504.9, 19.9) mm, rotated rx 0 ry 90 rz 0 deg; joints [-12.558, -28.465, 112.242, -16.576, -83.172, 51]
  Set speed (120.0 mm/s)
  MoveL 11536 to (495, 503.91, 19.9) mm, rotated rx 0 ry 90 rz 0 deg; joints [-12.467, -28.469, 112.268, -16.484, -83.19, 50.984]
  Set speed (15.0 mm/s)
  MoveL 11537 to (491.4, 500.31, 19.9) mm, rotated rx 0 ry 90 rz 0 deg; joints [-12.208, -28.548, 112.788, -16.208, -83.606, 50.833]
  Set speed (120.0 mm/s)
  MoveL 11538 to (491.4, 499.32, 19.9) mm, rotated rx 0 ry 90 rz 0 deg; joints [-12.116, -28.552, 112.814, -16.115, -83.624, 50.818]
  Set speed (15.0 mm/s)
  Call Extruder(0.168)
  MoveL 11539 to (495.48, 503.4, 19.9) mm, rotated rx 0 ry 90 rz 0 deg; joints [-12.41, -28.462, 112.225, -16.428, -83.153, 50.989]
  Set speed (120.0 mm/s)
  MoveL 11540 to (496.47, 503.4, 19.9) mm, rotated rx 0 ry 90 rz 0 deg; joints [-12.39, -28.444, 112.107, -16.411, -83.057, 51.015]
  Set speed (15.0 mm/s)
  Call Extruder(0.208)
  MoveL 11541 to (491.4, 498.33, 19.9) mm, rotated rx 0 ry 90 rz 0 deg; joints [-12.024, -28.556, 112.839, -16.022, -83.642, 50.804]
  Set speed (120.0 mm/s)
  MoveL 11542 to (491.4, 497.34, 19.9) mm, rotated rx 0 ry 90 rz 0 deg; joints [-11.932, -28.559, 112.864, -15.929, -83.659, 50.789]
  Set speed (15.0 mm/s)
  Call Extruder(0.249)
  MoveL 11543 to (497.46, 503.4, 19.9) mm, rotated rx 0 ry 90 rz 0 deg; joints [-12.37, -28.425, 111.989, -16.395, -82.961, 51.041]
  Set speed (120.0 mm/s)
  MoveL 11544 to (498.45, 503.4, 19.9) mm, rotated rx 0 ry 90 rz 0 deg; joints [-12.351, -28.406, 111.871, -16.378, -82.866, 51.067]
  Set speed (15.0 mm/s)
  Call Extruder(0.290)
  MoveL 11545 to (491.4, 496.35, 19.9) mm, rotated rx 0 ry 90 rz 0 deg; joints [-11.839, -28.563, 112.888, -15.835, -83.677, 50.774]
  Set speed (120.0 mm/s)
  MoveL 11546 to (491.4, 495.36, 19.9) mm, rotated rx 0 ry 90 rz 0 deg; joints [-11.747, -28.567, 112.913, -15.742, -83.695, 50.76]
  Set speed (15.0 mm/s)
  Call Extruder(0.321)
  MoveL 11547 to (499.2, 503.16, 19.9) mm, rotated rx 0 ry 90 rz 0 deg; joints [-12.313, -28.393, 111.788, -16.343, -82.797, 51.083]
  MoveL 11548 to (499.32, 503.28, 19.9) mm, rotated rx 0 ry 90 rz 0 deg; joints [-12.322, -28.39, 111.77, -16.352, -82.783, 51.088]
  Set speed (120.0 mm/s)
  MoveL 11549 to (498.17, 501.14, 19.9) mm, rotated rx 0 ry 90 rz 0 deg; joints [-12.149, -28.421, 111.964, -16.172, -82.934, 51.023]
  Set speed (15.0 mm/s)
  Call Extruder(0.278)
  MoveL 11550 to (491.4, 494.37, 19.9) mm, rotated rx 0 ry 90 rz 0 deg; joints [-11.655, -28.57, 112.937, -15.649, -83.712, 50.745]
  Set speed (120.0 mm/s)
  MoveL 11551 to (491.4, 493.38, 19.9) mm, rotated rx 0 ry 90 rz 0 deg; joints [-11.563, -28.574, 112.961, -15.555, -83.73, 50.731]
  Set speed (15.0 mm/s)
  Call Extruder(0.236)
  MoveL 11552 to (497.14, 499.12, 19.9) mm, rotated rx 0 ry 90 rz 0 deg; joints [-11.983, -28.448, 112.138, -16, -83.07, 50.964]
  MoveL 11553 to (497.26, 499.24, 19.9) mm, rotated rx 0 ry 90 rz 0 deg; joints [-11.992, -28.446, 112.12, -16.01, -83.056, 50.969]
  Set speed (120.0 mm/s)
  MoveL 11554 to (496.1, 497.09, 19.9) mm, rotated rx 0 ry 90 rz 0 deg; joints [-11.817, -28.475, 112.312, -15.828, -83.206, 50.906]
  Set speed (15.0 mm/s)
  Call Extruder(0.193)
  MoveL 11555 to (491.4, 492.39, 19.9) mm, rotated rx 0 ry 90 rz 0 deg; joints [-11.47, -28.577, 112.985, -15.462, -83.747, 50.717]
  Set speed (120.0 mm/s)
  MoveL 11556 to (491.4, 491.4, 19.9) mm, rotated rx 0 ry 90 rz 0 deg; joints [-11.378, -28.581, 113.009, -15.368, -83.764, 50.703]
  Set speed (15.0 mm/s)
  Call Extruder(0.151)
  MoveL 11557 to (495.07, 495.07, 19.9) mm, rotated rx 0 ry 90 rz 0 deg; joints [-11.65, -28.502, 112.484, -15.655, -83.342, 50.849]
  Set speed (120.0 mm/s)
  MoveL 11558 to (494.92, 493.93, 19.9) mm, rotated rx 0 ry 90 rz 0 deg; joints [-11.546, -28.509, 112.531, -15.55, -83.377, 50.828]
  Set speed (15.0 mm/s)
  Call Extruder(0.104)
  MoveL 11559 to (492.39, 491.4, 19.9) mm, rotated rx 0 ry 90 rz 0 deg; joints [-11.36, -28.563, 112.891, -15.353, -83.667, 50.728]
  Set speed (120.0 mm/s)
  MoveL 11560 to (493.38, 491.4, 19.9) mm, rotated rx 0 ry 90 rz 0 deg; joints [-11.341, -28.546, 112.774, -15.337, -83.57, 50.752]
  Set speed (15.0 mm/s)
  Call Extruder(0.063)
  MoveL 11561 to (494.92, 492.94, 19.9) mm, rotated rx 0 ry 90 rz 0 deg; joints [-11.455, -28.513, 112.555, -15.457, -83.394, 50.813]
  Set speed (120.0 mm/s)
  MoveL 11562 to (495.57, 492.6, 19.9) mm, rotated rx 0 ry 90 rz 0 deg; joints [-11.411, -28.502, 112.485, -15.415, -83.336, 50.825]
  Set speed (15.0 mm/s)
  Call Extruder(0.049)
  MoveL 11563 to (494.37, 491.4, 19.9) mm, rotated rx 0 ry 90 rz 0 deg; joints [-11.323, -28.528, 112.656, -15.321, -83.473, 50.777]
  Set speed (120.0 mm/s)
  MoveL 11564 to (495.36, 491.4, 19.9) mm, rotated rx 0 ry 90 rz 0 deg; joints [-11.304, -28.51, 112.538, -15.306, -83.376, 50.802]
  Set speed (15.0 mm/s)
  MoveL 11565 to (496.56, 492.6, 19.9) mm, rotated rx 0 ry 90 rz 0 deg; joints [-11.393, -28.484, 112.367, -15.4, -83.239, 50.85]
  Set speed (120.0 mm/s)
  MoveL 11566 to (497.55, 492.6, 19.9) mm, rotated rx 0 ry 90 rz 0 deg; joints [-11.374, -28.466, 112.249, -15.384, -83.142, 50.874]
  Set speed (15.0 mm/s)
  MoveL 11567 to (496.35, 491.4, 19.9) mm, rotated rx 0 ry 90 rz 0 deg; joints [-11.286, -28.492, 112.42, -15.291, -83.279, 50.827]
  Set speed (120.0 mm/s)
  MoveL 11568 to (497.34, 491.4, 19.9) mm, rotated rx 0 ry 90 rz 0 deg; joints [-11.268, -28.474, 112.302, -15.275, -83.182, 50.851]
  Set speed (15.0 mm/s)
  MoveL 11569 to (498.54, 492.6, 19.9) mm, rotated rx 0 ry 90 rz 0 deg; joints [-11.356, -28.447, 112.131, -15.369, -83.045, 50.899]
  Set speed (120.0 mm/s)
  MoveL 11570 to (499.53, 492.6, 19.9) mm, rotated rx 0 ry 90 rz 0 deg; joints [-11.338, -28.429, 112.012, -15.354, -82.949, 50.924]
  Set speed (15.0 mm/s)
  MoveL 11571 to (498.33, 491.4, 19.9) mm, rotated rx 0 ry 90 rz 0 deg; joints [-11.249, -28.456, 112.184, -15.26, -83.086, 50.876]
  Set speed (120.0 mm/s)
  MoveL 11572 to (499.32, 491.4, 19.9) mm, rotated rx 0 ry 90 rz 0 deg; joints [-11.231, -28.437, 112.066, -15.245, -82.989, 50.9]
  Set speed (15.0 mm/s)
  MoveL 11573 to (500.52, 492.6, 19.9) mm, rotated rx 0 ry 90 rz 0 deg; joints [-11.319, -28.41, 111.894, -15.339, -82.852, 50.948]
  Set speed (120.0 mm/s)
  MoveL 11574 to (501.51, 492.6, 19.9) mm, rotated rx 0 ry 90 rz 0 deg; joints [-11.301, -28.391, 111.775, -15.324, -82.755, 50.973]
  Set speed (15.0 mm/s)
  MoveL 11575 to (500.31, 491.4, 19.9) mm, rotated rx 0 ry 90 rz 0 deg; joints [-11.213, -28.418, 111.947, -15.23, -82.892, 50.925]
  Set speed (120.0 mm/s)
  MoveL 11576 to (501.3, 491.4, 19.9) mm, rotated rx 0 ry 90 rz 0 deg; joints [-11.195, -28.4, 111.829, -15.215, -82.795, 50.949]
  Set speed (15.0 mm/s)
  MoveL 11577 to (502.5, 492.6, 19.9) mm, rotated rx 0 ry 90 rz 0 deg; joints [-11.283, -28.372, 111.657, -15.309, -82.659, 50.997]
  Set speed (120.0 mm/s)
  MoveL 11578 to (503.49, 492.6, 19.9) mm, rotated rx 0 ry 90 rz 0 deg; joints [-11.265, -28.353, 111.538, -15.294, -82.562, 51.022]
  Set speed (15.0 mm/s)
  MoveL 11579 to (502.29, 491.4, 19.9) mm, rotated rx 0 ry 90 rz 0 deg; joints [-11.177, -28.38, 111.71, -15.2, -82.699, 50.973]
  Set speed (120.0 mm/s)
  MoveL 11580 to (503.28, 491.4, 19.9) mm, rotated rx 0 ry 90 rz 0 deg; joints [-11.159, -28.361, 111.591, -15.186, -82.602, 50.998]
  Set speed (15.0 mm/s)
  Call Extruder(0.049)
  MoveL 11581 to (504.48, 492.6, 19.9) mm, rotated rx 0 ry 90 rz 0 deg; joints [-11.247, -28.333, 111.419, -15.279, -82.466, 51.046]
  Set speed (120.0 mm/s)
  MoveL 11582 to (505.47, 492.6, 19.9) mm, rotated rx 0 ry 90 rz 0 deg; joints [-11.229, -28.314, 111.3, -15.265, -82.369, 51.07]
  Set speed (15.0 mm/s)
  MoveL 11583 to (504.27, 491.4, 19.9) mm, rotated rx 0 ry 90 rz 0 deg; joints [-11.141, -28.342, 111.472, -15.171, -82.505, 51.022]
  Set speed (120.0 mm/s)
  MoveL 11584 to (505.26, 491.4, 19.9) mm, rotated rx 0 ry 90 rz 0 deg; joints [-11.123, -28.322, 111.353, -15.157, -82.409, 51.046]
  Set speed (15.0 mm/s)
  Call Extruder(0.137)
  MoveL 11585 to (508.59, 494.74, 19.9) mm, rotated rx 0 ry 90 rz 0 deg; joints [-11.366, -28.242, 110.872, -15.416, -82.03, 51.182]
  Set speed (120.0 mm/s)
  MoveL 11586 to (508.59, 495.72, 19.9) mm, rotated rx 0 ry 90 rz 0 deg; joints [-11.456, -28.238, 110.848, -15.507, -82.014, 51.199]
  Set speed (15.0 mm/s)
  Call Extruder(0.127)
  MoveL 11587 to (505.52, 492.65, 19.9) mm, rotated rx 0 ry 90 rz 0 deg; joints [-11.232, -28.312, 111.293, -15.268, -82.364, 51.072]
  Set speed (120.0 mm/s)
  MoveL 11588 to (505.52, 493.64, 19.9) mm, rotated rx 0 ry 90 rz 0 deg; joints [-11.323, -28.309, 111.27, -15.36, -82.348, 51.088]
  Set speed (15.0 mm/s)
  MoveL 11589 to (508.59, 496.71, 19.9) mm, rotated rx 0 ry 90 rz 0 deg; joints [-11.546, -28.234, 110.824, -15.599, -81.998, 51.216]
  Set speed (120.0 mm/s)
  MoveL 11590 to (508.59, 497.7, 19.9) mm, rotated rx 0 ry 90 rz 0 deg; joints [-11.636, -28.23, 110.799, -15.69, -81.981, 51.232]
  Set speed (15.0 mm/s)
  MoveL 11591 to (505.52, 494.63, 19.9) mm, rotated rx 0 ry 90 rz 0 deg; joints [-11.413, -28.305, 111.246, -15.452, -82.331, 51.104]
  Set speed (120.0 mm/s)
  MoveL 11592 to (505.52, 495.62, 19.9) mm, rotated rx 0 ry 90 rz 0 deg; joints [-11.503, -28.301, 111.222, -15.543, -82.315, 51.121]
  Set speed (15.0 mm/s)
  MoveL 11593 to (508.59, 498.69, 19.9) mm, rotated rx 0 ry 90 rz 0 deg; joints [-11.725, -28.225, 110.775, -15.781, -81.965, 51.249]
  Set speed (120.0 mm/s)
  MoveL 11594 to (508.59, 499.68, 19.9) mm, rotated rx 0 ry 90 rz 0 deg; joints [-11.815, -28.221, 110.75, -15.872, -81.948, 51.266]
  Set speed (15.0 mm/s)
  MoveL 11595 to (505.52, 496.61, 19.9) mm, rotated rx 0 ry 90 rz 0 deg; joints [-11.593, -28.297, 111.197, -15.635, -82.298, 51.137]
  Set speed (120.0 mm/s)
  MoveL 11596 to (504.84, 496.93, 19.9) mm, rotated rx 0 ry 90 rz 0 deg; joints [-11.635, -28.309, 111.27, -15.675, -82.358, 51.125]
  Set speed (15.0 mm/s)
  Call Extruder(0.154)
  MoveL 11597 to (508.59, 500.67, 19.9) mm, rotated rx 0 ry 90 rz 0 deg; joints [-11.904, -28.217, 110.725, -15.964, -81.931, 51.283]
  Set speed (120.0 mm/s)
  MoveL 11598 to (508.59, 501.66, 19.9) mm, rotated rx 0 ry 90 rz 0 deg; joints [-11.994, -28.212, 110.699, -16.055, -81.914, 51.301]
  Set speed (15.0 mm/s)
  Call Extruder(0.195)
  MoveL 11599 to (503.85, 496.93, 19.9) mm, rotated rx 0 ry 90 rz 0 deg; joints [-11.654, -28.328, 111.389, -15.69, -82.454, 51.101]
  Set speed (120.0 mm/s)
  MoveL 11600 to (502.87, 496.93, 19.9) mm, rotated rx 0 ry 90 rz 0 deg; joints [-11.672, -28.348, 111.508, -15.705, -82.551, 51.076]
  Set speed (15.0 mm/s)
  Call Extruder(0.236)
  MoveL 11601 to (508.59, 502.65, 19.9) mm, rotated rx 0 ry 90 rz 0 deg; joints [-12.083, -28.208, 110.674, -16.146, -81.897, 51.318]
  Set speed (120.0 mm/s)
  MoveL 11602 to (508.59, 503.64, 19.9) mm, rotated rx 0 ry 90 rz 0 deg; joints [-12.172, -28.204, 110.648, -16.237, -81.88, 51.335]
  Set speed (15.0 mm/s)
  Call Extruder(0.277)
  MoveL 11603 to (501.88, 496.93, 19.9) mm, rotated rx 0 ry 90 rz 0 deg; joints [-11.691, -28.367, 111.626, -15.721, -82.647, 51.051]
  Set speed (120.0 mm/s)
  MoveL 11604 to (500.94, 496.98, 19.9) mm, rotated rx 0 ry 90 rz 0 deg; joints [-11.714, -28.385, 111.737, -15.74, -82.737, 51.028]
  Set speed (15.0 mm/s)
  Call Extruder(0.315)
  MoveL 11605 to (508.59, 504.63, 19.9) mm, rotated rx 0 ry 90 rz 0 deg; joints [-12.262, -28.199, 110.622, -16.328, -81.863, 51.353]
  Set speed (120.0 mm/s)
  MoveL 11606 to (508.59, 505.62, 19.9) mm, rotated rx 0 ry 90 rz 0 deg; joints [-12.351, -28.195, 110.596, -16.419, -81.845, 51.37]
  Set speed (15.0 mm/s)
  Call Extruder(0.272)
  MoveL 11607 to (501.98, 499.01, 19.9) mm, rotated rx 0 ry 90 rz 0 deg; joints [-11.879, -28.357, 111.562, -15.913, -82.601, 51.087]
  MoveL 11608 to (501.85, 498.88, 19.9) mm, rotated rx 0 ry 90 rz 0 deg; joints [-11.871, -28.359, 111.58, -15.903, -82.615, 51.082]
  Set speed (120.0 mm/s)
  MoveL 11609 to (503.02, 501.04, 19.9) mm, rotated rx 0 ry 90 rz 0 deg; joints [-12.044, -28.328, 111.386, -16.084, -82.465, 51.147]
  Set speed (15.0 mm/s)
  Call Extruder(0.230)
  MoveL 11610 to (508.59, 506.61, 19.9) mm, rotated rx 0 ry 90 rz 0 deg; joints [-12.44, -28.19, 110.57, -16.51, -81.828, 51.388]
  Set speed (120.0 mm/s)
  MoveL 11611 to (508.59, 507.6, 19.9) mm, rotated rx 0 ry 90 rz 0 deg; joints [-12.529, -28.186, 110.544, -16.6, -81.81, 51.406]
  Set speed (15.0 mm/s)
  Call Extruder(0.187)
  MoveL 11612 to (504.05, 503.06, 19.9) mm, rotated rx 0 ry 90 rz 0 deg; joints [-12.209, -28.299, 111.209, -16.255, -82.329, 51.208]
  MoveL 11613 to (503.93, 502.94, 19.9) mm, rotated rx 0 ry 90 rz 0 deg; joints [-12.2, -28.302, 111.227, -16.246, -82.343, 51.203]
  Set speed (120.0 mm/s)
  MoveL 11614 to (505.09, 505.09, 19.9) mm, rotated rx 0 ry 90 rz 0 deg; joints [-12.372, -28.269, 111.032, -16.426, -82.193, 51.27]
  Set speed (15.0 mm/s)
  Call Extruder(0.144)
  MoveL 11615 to (508.59, 508.59, 19.9) mm, rotated rx 0 ry 90 rz 0 deg; joints [-12.618, -28.181, 110.517, -16.691, -81.793, 51.423]
  Set speed (120.0 mm/s)
  MoveL 11616 to (507.6, 508.59, 19.9) mm, rotated rx 0 ry 90 rz 0 deg; joints [-12.638, -28.202, 110.636, -16.707, -81.888, 51.397]
  Set speed (15.0 mm/s)
  Call Extruder(0.094)
  MoveL 11617 to (505.33, 506.32, 19.9) mm, rotated rx 0 ry 90 rz 0 deg; joints [-12.479, -28.259, 110.97, -16.535, -82.148, 51.297]
  Set speed (120.0 mm/s)
  MoveL 11618 to (505.33, 507.31, 19.9) mm, rotated rx 0 ry 90 rz 0 deg; joints [-12.568, -28.254, 110.944, -16.626, -82.13, 51.315]
  Set speed (15.0 mm/s)
  Call Extruder(0.053)
  MoveL 11619 to (506.61, 508.59, 19.9) mm, rotated rx 0 ry 90 rz 0 deg; joints [-12.658, -28.222, 110.755, -16.723, -81.983, 51.371]
  Set speed (120.0 mm/s)
  MoveL 11620 to (505.62, 508.59, 19.9) mm, rotated rx 0 ry 90 rz 0 deg; joints [-12.678, -28.242, 110.874, -16.74, -82.078, 51.345]
  Set speed (15.0 mm/s)
  Call Extruder(0.036)
  MoveL 11621 to (504.75, 507.72, 19.9) mm, rotated rx 0 ry 90 rz 0 deg; joints [-12.617, -28.264, 111.003, -16.674, -82.178, 51.307]
  Set speed (120.0 mm/s)
  MoveL 11622 to (504.63, 508.59, 19.9) mm, rotated rx 0 ry 90 rz 0 deg; joints [-12.698, -28.262, 110.993, -16.756, -82.174, 51.319]
  Set speed (15.0 mm/s)
  MoveL 11623 to (503.76, 507.72, 19.9) mm, rotated rx 0 ry 90 rz 0 deg; joints [-12.637, -28.284, 111.121, -16.69, -82.274, 51.28]
  Set speed (120.0 mm/s)
  MoveL 11624 to (503.64, 508.59, 19.9) mm, rotated rx 0 ry 90 rz 0 deg; joints [-12.719, -28.282, 111.112, -16.772, -82.269, 51.292]
  Set speed (15.0 mm/s)
  MoveL 11625 to (502.77, 507.72, 19.9) mm, rotated rx 0 ry 90 rz 0 deg; joints [-12.657, -28.304, 111.24, -16.707, -82.369, 51.254]
  Set speed (120.0 mm/s)
  MoveL 11626 to (502.65, 508.59, 19.9) mm, rotated rx 0 ry 90 rz 0 deg; joints [-12.739, -28.302, 111.231, -16.789, -82.365, 51.266]
  Set speed (15.0 mm/s)
  MoveL 11627 to (501.78, 507.72, 19.9) mm, rotated rx 0 ry 90 rz 0 deg; joints [-12.678, -28.323, 111.358, -16.723, -82.465, 51.228]
  Set speed (120.0 mm/s)
  MoveL 11628 to (501.66, 508.59, 19.9) mm, rotated rx 0 ry 90 rz 0 deg; joints [-12.759, -28.322, 111.349, -16.806, -82.46, 51.24]
  Set speed (15.0 mm/s)
  MoveL 11629 to (500.79, 507.72, 19.9) mm, rotated rx 0 ry 90 rz 0 deg; joints [-12.698, -28.343, 111.477, -16.74, -82.56, 51.201]
  Set speed (120.0 mm/s)
  MoveL 11630 to (500.67, 508.59, 19.9) mm, rotated rx 0 ry 90 rz 0 deg; joints [-12.78, -28.341, 111.467, -16.823, -82.555, 51.213]
  Set speed (15.0 mm/s)
  MoveL 11631 to (499.8, 507.72, 19.9) mm, rotated rx 0 ry 90 rz 0 deg; joints [-12.718, -28.362, 111.595, -16.757, -82.656, 51.175]
  Set speed (120.0 mm/s)
  MoveL 11632 to (499.68, 508.59, 19.9) mm, rotated rx 0 ry 90 rz 0 deg; joints [-12.8, -28.36, 111.586, -16.839, -82.651, 51.187]
  Set speed (15.0 mm/s)
  MoveL 11633 to (498.81, 507.72, 19.9) mm, rotated rx 0 ry 90 rz 0 deg; joints [-12.739, -28.381, 111.713, -16.774, -82.751, 51.148]
  Set speed (120.0 mm/s)
  MoveL 11634 to (498.69, 508.59, 19.9) mm, rotated rx 0 ry 90 rz 0 deg; joints [-12.821, -28.379, 111.704, -16.856, -82.746, 51.16]
  Set speed (15.0 mm/s)
  MoveL 11635 to (497.82, 507.72, 19.9) mm, rotated rx 0 ry 90 rz 0 deg; joints [-12.759, -28.4, 111.831, -16.791, -82.847, 51.122]
  Set speed (120.0 mm/s)
  MoveL 11636 to (497.7, 508.59, 19.9) mm, rotated rx 0 ry 90 rz 0 deg; joints [-12.841, -28.398, 111.822, -16.874, -82.842, 51.133]
  Set speed (15.0 mm/s)
  Call Extruder(0.036)
  MoveL 11637 to (496.83, 507.72, 19.9) mm, rotated rx 0 ry 90 rz 0 deg; joints [-12.779, -28.419, 111.949, -16.808, -82.942, 51.095]
  Set speed (120.0 mm/s)
  MoveL 11638 to (496.71, 508.59, 19.9) mm, rotated rx 0 ry 90 rz 0 deg; joints [-12.862, -28.417, 111.94, -16.891, -82.937, 51.107]
  Set speed (15.0 mm/s)
  MoveL 11639 to (495.84, 507.72, 19.9) mm, rotated rx 0 ry 90 rz 0 deg; joints [-12.8, -28.437, 112.067, -16.825, -83.038, 51.069]
  Set speed (120.0 mm/s)
  MoveL 11640 to (504.35, 506.75, 19.9) mm, rotated rx 0 ry 90 rz 0 deg; joints [-12.537, -28.276, 111.076, -16.59, -82.234, 51.279]
  Set speed (1000.0 mm/s)
  MoveL 11641 to (508.59, 493.75, 19.9) mm, rotated rx 0 ry 90 rz 0 deg; joints [-11.277, -28.246, 110.896, -15.325, -82.046, 51.166]
  Set speed (15.0 mm/s)
  Call Extruder(0.096)
  MoveL 11642 to (506.25, 491.4, 19.9) mm, rotated rx 0 ry 90 rz 0 deg; joints [-11.106, -28.303, 111.234, -15.142, -82.312, 51.07]
  Set speed (120.0 mm/s)
  MoveL 11643 to (507.24, 491.4, 19.9) mm, rotated rx 0 ry 90 rz 0 deg; joints [-11.088, -28.283, 111.115, -15.128, -82.216, 51.094]
  Set speed (15.0 mm/s)
  Call Extruder(0.056)
  MoveL 11644 to (508.59, 492.76, 19.9) mm, rotated rx 0 ry 90 rz 0 deg; joints [-11.187, -28.25, 110.92, -15.233, -82.062, 51.149]
  Set speed (120.0 mm/s)
  MoveL 11645 to (508.59, 491.76, 19.9) mm, rotated rx 0 ry 90 rz 0 deg; joints [-11.097, -28.254, 110.943, -15.142, -82.078, 51.133]
  Set speed (15.0 mm/s)
  Call Extruder(0.015)
  MoveL 11646 to (508.23, 491.4, 19.9) mm, rotated rx 0 ry 90 rz 0 deg; joints [-11.07, -28.263, 110.995, -15.114, -82.119, 51.118]
  Set speed (120.0 mm/s)
  MoveL 11647 to (495.89, 493.58, 19.9) mm, rotated rx 0 ry 90 rz 0 deg; joints [-11.496, -28.493, 112.423, -15.502, -83.287, 50.848]
  Set speed (1000.0 mm/s)
  MoveL 11648 to (490.47, 509.53, 19.9) mm, rotated rx 0 ry 90 rz 0 deg; joints [-13.08, -28.528, 112.654, -17.089, -83.522, 50.951]
  Set speed (1000.0 mm/s)
  MoveL 11649 to (490.4, 509.6, 19.9) mm, rotated rx 0 ry 90 rz 0 deg; joints [-13.088, -28.529, 112.661, -17.097, -83.527, 50.951]
  Set speed (1000.0 mm/s)
  MoveL 11650 to (490.4, 509.6, 20) mm, rotated rx 0 ry 90 rz 0 deg; joints [-13.088, -28.539, 112.666, -17.097, -83.522, 50.952]
  Set speed (15.0 mm/s)
  Call Extruder(0.559)
  MoveL 11651 to (490.4, 490.4, 20) mm, rotated rx 0 ry 90 rz 0 deg; joints [-11.303, -28.612, 113.157, -15.29, -83.874, 50.665]
  MoveL 11652 to (509.6, 490.4, 20) mm, rotated rx 0 ry 90 rz 0 deg; joints [-10.955, -28.249, 110.859, -15.002, -81.996, 51.136]
  MoveL 11653 to (509.6, 509.6, 20) mm, rotated rx 0 ry 90 rz 0 deg; joints [-12.688, -28.166, 110.373, -16.767, -81.673, 51.47]
  MoveL 11654 to (490.4, 509.6, 20) mm, rotated rx 0 ry 90 rz 0 deg; joints [-13.088, -28.539, 112.666, -17.097, -83.522, 50.952]
  Set speed (120.0 mm/s)
  MoveL 11655 to (490.4, 509.2, 20) mm, rotated rx 0 ry 90 rz 0 deg; joints [-13.051, -28.541, 112.677, -17.06, -83.53, 50.946]
  Set speed (1000.0 mm/s)
  MoveL 11656 to (490.5, 509.2, 20) mm, rotated rx 0 ry 90 rz 0 deg; joints [-13.049, -28.539, 112.665, -17.058, -83.52, 50.949]
  Set speed (1000.0 mm/s)
  MoveL 11657 to (495.94, 504.34, 20) mm, rotated rx 0 ry 90 rz 0 deg; joints [-12.487, -28.46, 112.151, -16.508, -83.086, 51.018]
  Set speed (1000.0 mm/s)
  MoveL 11658 to (496.01, 504.41, 20) mm, rotated rx 0 ry 90 rz 0 deg; joints [-12.492, -28.459, 112.141, -16.513, -83.078, 51.021]
  Set speed (15.0 mm/s)
  Call Extruder(0.067)
  MoveL 11659 to (496.01, 506.72, 20) mm, rotated rx 0 ry 90 rz 0 deg; joints [-12.705, -28.449, 112.079, -16.729, -83.035, 51.058]
  Call Extruder(0.242)
  MoveL 11660 to (504.33, 506.72, 20) mm, rotated rx 0 ry 90 rz 0 deg; joints [-12.535, -28.288, 111.085, -16.588, -82.232, 51.279]
  Call Extruder(0.027)
  MoveL 11661 to (504.33, 505.8, 20) mm, rotated rx 0 ry 90 rz 0 deg; joints [-12.452, -28.292, 111.11, -16.504, -82.249, 51.264]
  Call Extruder(0.306)
  MoveL 11662 to (499.53, 496.43, 20) mm, rotated rx 0 ry 90 rz 0 deg; joints [-11.69, -28.425, 111.924, -15.711, -82.878, 50.985]
  Call Extruder(0.017)
  MoveL 11663 to (499.27, 495.92, 20) mm, rotated rx 0 ry 90 rz 0 deg; joints [-11.648, -28.431, 111.968, -15.668, -82.912, 50.97]
  Call Extruder(0.010)
  MoveL 11664 to (499.84, 495.92, 20) mm, rotated rx 0 ry 90 rz 0 deg; joints [-11.637, -28.421, 111.9, -15.659, -82.857, 50.985]
  Call Extruder(0.000)
  MoveL 11665 to (499.84, 495.92, 20) mm, rotated rx 0 ry 90 rz 0 deg; joints [-11.637, -28.421, 111.9, -15.659, -82.857, 50.985]
  Call Extruder(0.136)
  MoveL 11666 to (504.51, 495.92, 20) mm, rotated rx 0 ry 90 rz 0 deg; joints [-11.55, -28.33, 111.34, -15.587, -82.402, 51.102]
  Call Extruder(0.067)
  MoveL 11667 to (504.51, 493.61, 20) mm, rotated rx 0 ry 90 rz 0 deg; joints [-11.338, -28.339, 111.396, -15.372, -82.441, 51.065]
  Call Extruder(0.250)
  MoveL 11668 to (495.92, 493.61, 20) mm, rotated rx 0 ry 90 rz 0 deg; joints [-11.498, -28.503, 112.424, -15.504, -83.279, 50.85]
  Call Extruder(0.027)
  MoveL 11669 to (495.92, 494.52, 20) mm, rotated rx 0 ry 90 rz 0 deg; joints [-11.583, -28.499, 112.402, -15.59, -83.263, 50.864]
  Call Extruder(0.306)
  MoveL 11670 to (500.7, 503.9, 20) mm, rotated rx 0 ry 90 rz 0 deg; joints [-12.351, -28.371, 111.594, -16.387, -82.633, 51.136]
  Call Extruder(0.017)
  MoveL 11671 to (500.96, 504.41, 20) mm, rotated rx 0 ry 90 rz 0 deg; joints [-12.392, -28.364, 111.55, -16.43, -82.599, 51.151]
  Call Extruder(0.010)
  MoveL 11672 to (500.39, 504.41, 20) mm, rotated rx 0 ry 90 rz 0 deg; joints [-12.404, -28.375, 111.618, -16.439, -82.654, 51.137]
  Call Extruder(0.000)
  MoveL 11673 to (500.39, 504.4, 20) mm, rotated rx 0 ry 90 rz 0 deg; joints [-12.404, -28.375, 111.618, -16.439, -82.654, 51.136]
  Call Extruder(0.128)
  MoveL 11674 to (496.01, 504.41, 20) mm, rotated rx 0 ry 90 rz 0 deg; joints [-12.492, -28.459, 112.141, -16.513, -83.078, 51.021]
  Set speed (120.0 mm/s)
  MoveL 11675 to (496.01, 504.8, 20) mm, rotated rx 0 ry 90 rz 0 deg; joints [-12.529, -28.457, 112.13, -16.55, -83.071, 51.027]
  Set speed (1000.0 mm/s)
  MoveL 11676 to (495.91, 504.81, 20) mm, rotated rx 0 ry 90 rz 0 deg; joints [-12.531, -28.459, 112.142, -16.552, -83.081, 51.024]
  Set speed (1000.0 mm/s)
  MoveL 11677 to (495.32, 503.72, 20) mm, rotated rx 0 ry 90 rz 0 deg; joints [-12.443, -28.474, 112.241, -16.46, -83.158, 50.991]
  Set speed (15.0 mm/s)
  Call Extruder(0.107)
  MoveL 11678 to (495.32, 507.41, 20) mm, rotated rx 0 ry 90 rz 0 deg; joints [-12.782, -28.459, 112.143, -16.805, -83.089, 51.051]
  Call Extruder(0.282)
  MoveL 11679 to (505.02, 507.41, 20) mm, rotated rx 0 ry 90 rz 0 deg; joints [-12.583, -28.271, 110.984, -16.641, -82.153, 51.31]
  Call Extruder(0.052)
  MoveL 11680 to (505.02, 505.64, 20) mm, rotated rx 0 ry 90 rz 0 deg; joints [-12.423, -28.278, 111.031, -16.477, -82.185, 51.279]
  Call Extruder(0.295)
  MoveL 11681 to (500.4, 496.61, 20) mm, rotated rx 0 ry 90 rz 0 deg; joints [-11.69, -28.407, 111.816, -15.715, -82.791, 51.01]
  Call Extruder(0.140)
  MoveL 11682 to (505.2, 496.61, 20) mm, rotated rx 0 ry 90 rz 0 deg; joints [-11.6, -28.313, 111.24, -15.64, -82.324, 51.131]
  Call Extruder(0.107)
  MoveL 11683 to (505.2, 492.92, 20) mm, rotated rx 0 ry 90 rz 0 deg; joints [-11.263, -28.328, 111.33, -15.298, -82.385, 51.07]
  Call Extruder(0.290)
  MoveL 11684 to (495.23, 492.92, 20) mm, rotated rx 0 ry 90 rz 0 deg; joints [-11.447, -28.518, 112.523, -15.45, -83.358, 50.823]
  Call Extruder(0.052)
  MoveL 11685 to (495.23, 494.69, 20) mm, rotated rx 0 ry 90 rz 0 deg; joints [-11.611, -28.511, 112.48, -15.617, -83.327, 50.849]
  Call Extruder(0.295)
  MoveL 11686 to (499.84, 503.72, 20) mm, rotated rx 0 ry 90 rz 0 deg; joints [-12.352, -28.389, 111.702, -16.385, -82.72, 51.11]
  Call Extruder(0.132)
  MoveL 11687 to (495.32, 503.72, 20) mm, rotated rx 0 ry 90 rz 0 deg; joints [-12.443, -28.474, 112.241, -16.46, -83.158, 50.991]
  Set speed (120.0 mm/s)
  MoveL 11688 to (491.09, 508.91, 20) mm, rotated rx 0 ry 90 rz 0 deg; joints [-13.01, -28.53, 112.603, -17.02, -83.469, 50.96]
  Set speed (15.0 mm/s)
  Call Extruder(0.519)
  MoveL 11689 to (491.09, 491.09, 20) mm, rotated rx 0 ry 90 rz 0 deg; joints [-11.355, -28.598, 113.059, -15.344, -83.795, 50.692]
  MoveL 11690 to (508.91, 491.09, 20) mm, rotated rx 0 ry 90 rz 0 deg; joints [-11.03, -28.261, 110.926, -15.075, -82.053, 51.131]
  MoveL 11691 to (508.91, 508.91, 20) mm, rotated rx 0 ry 90 rz 0 deg; joints [-12.64, -28.183, 110.475, -16.715, -81.751, 51.439]
  MoveL 11692 to (491.09, 508.91, 20) mm, rotated rx 0 ry 90 rz 0 deg; joints [-13.01, -28.53, 112.603, -17.02, -83.469, 50.96]
  Set speed (120.0 mm/s)
  MoveL 11693 to (491.4, 491.62, 20) mm, rotated rx 0 ry 90 rz 0 deg; joints [-11.398, -28.591, 113.009, -15.389, -83.755, 50.707]
  Set speed (15.0 mm/s)
  Call Extruder(0.009)
  MoveL 11694 to (491.62, 491.4, 20) mm, rotated rx 0 ry 90 rz 0 deg; joints [-11.374, -28.588, 112.989, -15.365, -83.738, 50.709]
  Set speed (120.0 mm/s)
  MoveL 11695 to (492.61, 491.4, 20) mm, rotated rx 0 ry 90 rz 0 deg; joints [-11.356, -28.57, 112.871, -15.35, -83.641, 50.734]
  Set speed (15.0 mm/s)
  Call Extruder(0.049)
  MoveL 11696 to (491.4, 492.61, 20) mm, rotated rx 0 ry 90 rz 0 deg; joints [-11.49, -28.587, 112.985, -15.482, -83.738, 50.721]
  Set speed (120.0 mm/s)
  MoveL 11697 to (491.4, 493.6, 20) mm, rotated rx 0 ry 90 rz 0 deg; joints [-11.583, -28.584, 112.961, -15.575, -83.721, 50.736]
  Set speed (15.0 mm/s)
  Call Extruder(0.090)
  MoveL 11698 to (493.6, 491.4, 20) mm, rotated rx 0 ry 90 rz 0 deg; joints [-11.337, -28.553, 112.754, -15.334, -83.544, 50.759]
  Set speed (120.0 mm/s)
  MoveL 11699 to (494.58, 491.4, 20) mm, rotated rx 0 ry 90 rz 0 deg; joints [-11.319, -28.535, 112.636, -15.318, -83.447, 50.784]
  Set speed (15.0 mm/s)
  Call Extruder(0.131)
  MoveL 11700 to (491.4, 494.58, 20) mm, rotated rx 0 ry 90 rz 0 deg; joints [-11.675, -28.58, 112.937, -15.669, -83.703, 50.75]
  Set speed (120.0 mm/s)
  MoveL 11701 to (491.4, 495.58, 20) mm, rotated rx 0 ry 90 rz 0 deg; joints [-11.767, -28.576, 112.913, -15.762, -83.686, 50.764]
  Set speed (15.0 mm/s)
  Call Extruder(0.172)
  MoveL 11702 to (495.58, 491.4, 20) mm, rotated rx 0 ry 90 rz 0 deg; joints [-11.3, -28.517, 112.518, -15.303, -83.35, 50.809]
  Set speed (120.0 mm/s)
  MoveL 11703 to (496.57, 491.4, 20) mm, rotated rx 0 ry 90 rz 0 deg; joints [-11.282, -28.499, 112.4, -15.288, -83.253, 50.833]
  Set speed (15.0 mm/s)
  Call Extruder(0.049)
  MoveL 11704 to (495.37, 492.6, 20) mm, rotated rx 0 ry 90 rz 0 deg; joints [-11.415, -28.516, 112.514, -15.419, -83.35, 50.821]
  Set speed (120.0 mm/s)
  MoveL 11705 to (494.92, 493.05, 20) mm, rotated rx 0 ry 90 rz 0 deg; joints [-11.466, -28.523, 112.557, -15.468, -83.386, 50.817]
  Set speed (15.0 mm/s)
  Call Extruder(0.145)
  MoveL 11706 to (491.4, 496.56, 20) mm, rotated rx 0 ry 90 rz 0 deg; joints [-11.859, -28.573, 112.888, -15.856, -83.668, 50.779]
  Set speed (120.0 mm/s)
  MoveL 11707 to (491.4, 497.55, 20) mm, rotated rx 0 ry 90 rz 0 deg; joints [-11.951, -28.569, 112.863, -15.949, -83.65, 50.794]
  Set speed (15.0 mm/s)
  Call Extruder(0.145)
  MoveL 11708 to (494.92, 494.04, 20) mm, rotated rx 0 ry 90 rz 0 deg; joints [-11.557, -28.519, 112.533, -15.561, -83.369, 50.831]
  Set speed (120.0 mm/s)
  MoveL 11709 to (495.01, 494.94, 20) mm, rotated rx 0 ry 90 rz 0 deg; joints [-11.639, -28.514, 112.501, -15.644, -83.345, 50.847]
  Set speed (15.0 mm/s)
  Call Extruder(0.148)
  MoveL 11710 to (491.4, 498.54, 20) mm, rotated rx 0 ry 90 rz 0 deg; joints [-12.043, -28.565, 112.839, -16.042, -83.632, 50.808]
  Set speed (120.0 mm/s)
  MoveL 11711 to (491.4, 499.53, 20) mm, rotated rx 0 ry 90 rz 0 deg; joints [-12.135, -28.562, 112.813, -16.135, -83.614, 50.823]
  Set speed (15.0 mm/s)
  Call Extruder(0.162)
  MoveL 11712 to (495.34, 495.6, 20) mm, rotated rx 0 ry 90 rz 0 deg; joints [-11.693, -28.506, 112.445, -15.7, -83.301, 50.866]
  Set speed (120.0 mm/s)
  MoveL 11713 to (495.68, 496.25, 20) mm, rotated rx 0 ry 90 rz 0 deg; joints [-11.747, -28.497, 112.389, -15.756, -83.257, 50.884]
  Set speed (15.0 mm/s)
  Call Extruder(0.176)
  MoveL 11714 to (491.4, 500.52, 20) mm, rotated rx 0 ry 90 rz 0 deg; joints [-12.227, -28.558, 112.788, -16.228, -83.596, 50.838]
  Set speed (120.0 mm/s)
  MoveL 11715 to (491.4, 501.51, 20) mm, rotated rx 0 ry 90 rz 0 deg; joints [-12.319, -28.554, 112.763, -16.321, -83.578, 50.853]
  Set speed (15.0 mm/s)
  Call Extruder(0.190)
  MoveL 11716 to (496.01, 496.91, 20) mm, rotated rx 0 ry 90 rz 0 deg; joints [-11.802, -28.489, 112.333, -15.812, -83.213, 50.903]
  Set speed (120.0 mm/s)
  MoveL 11717 to (496.34, 497.56, 20) mm, rotated rx 0 ry 90 rz 0 deg; joints [-11.856, -28.48, 112.276, -15.868, -83.169, 50.921]
  Set speed (15.0 mm/s)
  Call Extruder(0.203)
  MoveL 11718 to (491.4, 502.5, 20) mm, rotated rx 0 ry 90 rz 0 deg; joints [-12.411, -28.55, 112.737, -16.414, -83.56, 50.868]
  Set speed (120.0 mm/s)
  MoveL 11719 to (491.4, 503.49, 20) mm, rotated rx 0 ry 90 rz 0 deg; joints [-12.502, -28.546, 112.711, -16.507, -83.541, 50.884]
  Set speed (15.0 mm/s)
  Call Extruder(0.217)
  MoveL 11720 to (496.68, 498.22, 20) mm, rotated rx 0 ry 90 rz 0 deg; joints [-11.91, -28.471, 112.22, -15.924, -83.125, 50.94]
  Set speed (120.0 mm/s)
  MoveL 11721 to (497.01, 498.88, 20) mm, rotated rx 0 ry 90 rz 0 deg; joints [-11.964, -28.462, 112.164, -15.98, -83.081, 50.959]
  Set speed (15.0 mm/s)
  Call Extruder(0.231)
  MoveL 11722 to (491.4, 504.48, 20) mm, rotated rx 0 ry 90 rz 0 deg; joints [-12.594, -28.542, 112.685, -16.6, -83.523, 50.899]
  Set speed (120.0 mm/s)
  MoveL 11723 to (491.4, 505.47, 20) mm, rotated rx 0 ry 90 rz 0 deg; joints [-12.686, -28.538, 112.659, -16.693, -83.504, 50.914]
  Set speed (15.0 mm/s)
  Call Extruder(0.245)
  MoveL 11724 to (497.35, 499.53, 20) mm, rotated rx 0 ry 90 rz 0 deg; joints [-12.017, -28.453, 112.107, -16.036, -83.036, 50.978]
  Set speed (120.0 mm/s)
  MoveL 11725 to (497.68, 500.19, 20) mm, rotated rx 0 ry 90 rz 0 deg; joints [-12.071, -28.445, 112.051, -16.092, -82.992, 50.997]
  Set speed (15.0 mm/s)
  Call Extruder(0.258)
  MoveL 11726 to (491.4, 506.46, 20) mm, rotated rx 0 ry 90 rz 0 deg; joints [-12.777, -28.534, 112.632, -16.786, -83.485, 50.93]
  Set speed (120.0 mm/s)
  MoveL 11727 to (491.4, 507.45, 20) mm, rotated rx 0 ry 90 rz 0 deg; joints [-12.868, -28.53, 112.605, -16.878, -83.466, 50.946]
  Set speed (15.0 mm/s)
  Call Extruder(0.148)
  MoveL 11728 to (495, 503.86, 20) mm, rotated rx 0 ry 90 rz 0 deg; joints [-12.462, -28.48, 112.275, -16.479, -83.186, 50.985]
  Set speed (120.0 mm/s)
  MoveL 11729 to (495.46, 503.4, 20) mm, rotated rx 0 ry 90 rz 0 deg; joints [-12.411, -28.473, 112.232, -16.428, -83.15, 50.99]
  Set speed (15.0 mm/s)
  Call Extruder(0.105)
  MoveL 11730 to (498.02, 500.84, 20) mm, rotated rx 0 ry 90 rz 0 deg; joints [-12.125, -28.436, 111.994, -16.147, -82.948, 51.016]
  Set speed (120.0 mm/s)
  MoveL 11731 to (498.35, 501.5, 20) mm, rotated rx 0 ry 90 rz 0 deg; joints [-12.178, -28.427, 111.937, -16.203, -82.904, 51.035]
  Set speed (15.0 mm/s)
  Call Extruder(0.078)
  MoveL 11732 to (496.45, 503.4, 20) mm, rotated rx 0 ry 90 rz 0 deg; joints [-12.391, -28.455, 112.115, -16.412, -83.054, 51.016]
  Set speed (120.0 mm/s)
  MoveL 11733 to (497.44, 503.4, 20) mm, rotated rx 0 ry 90 rz 0 deg; joints [-12.371, -28.436, 111.997, -16.395, -82.958, 51.042]
  Set speed (15.0 mm/s)
  Call Extruder(0.051)
  MoveL 11734 to (498.68, 502.15, 20) mm, rotated rx 0 ry 90 rz 0 deg; joints [-12.232, -28.418, 111.881, -16.258, -82.86, 51.055]
  Set speed (120.0 mm/s)
  MoveL 11735 to (499.02, 502.81, 20) mm, rotated rx 0 ry 90 rz 0 deg; joints [-12.285, -28.408, 111.824, -16.314, -82.816, 51.074]
  Set speed (15.0 mm/s)
  Call Extruder(0.024)
  MoveL 11736 to (498.43, 503.4, 20) mm, rotated rx 0 ry 90 rz 0 deg; joints [-12.351, -28.417, 111.879, -16.379, -82.862, 51.068]
  Set speed (120.0 mm/s)
  MoveL 11737 to (496.45, 504.19, 20) mm, rotated rx 0 ry 90 rz 0 deg; joints [-12.464, -28.451, 112.094, -16.486, -83.04, 51.029]
  Set speed (1000.0 mm/s)
  MoveL 11738 to (495, 504.85, 20) mm, rotated rx 0 ry 90 rz 0 deg; joints [-12.554, -28.476, 112.249, -16.572, -83.168, 51.001]
  Set speed (15.0 mm/s)
  Call Extruder(0.148)
  MoveL 11739 to (491.4, 508.44, 20) mm, rotated rx 0 ry 90 rz 0 deg; joints [-12.96, -28.526, 112.579, -16.971, -83.447, 50.961]
  Set speed (120.0 mm/s)
  MoveL 11740 to (492.24, 508.59, 20) mm, rotated rx 0 ry 90 rz 0 deg; joints [-12.956, -28.51, 112.475, -16.97, -83.363, 50.987]
  Set speed (15.0 mm/s)
  Call Extruder(0.113)
  MoveL 11741 to (495, 505.84, 20) mm, rotated rx 0 ry 90 rz 0 deg; joints [-12.645, -28.471, 112.223, -16.664, -83.149, 51.017]
  Set speed (120.0 mm/s)
  MoveL 11742 to (495, 506.83, 20) mm, rotated rx 0 ry 90 rz 0 deg; joints [-12.735, -28.467, 112.196, -16.756, -83.131, 51.033]
  Set speed (15.0 mm/s)
  Call Extruder(0.073)
  MoveL 11743 to (493.23, 508.59, 20) mm, rotated rx 0 ry 90 rz 0 deg; joints [-12.935, -28.492, 112.358, -16.952, -83.268, 51.014]
  Set speed (120.0 mm/s)
  MoveL 11744 to (494.22, 508.59, 20) mm, rotated rx 0 ry 90 rz 0 deg; joints [-12.914, -28.474, 112.24, -16.935, -83.172, 51.041]
  Set speed (15.0 mm/s)
  Call Extruder(0.036)
  MoveL 11745 to (495.1, 507.72, 20) mm, rotated rx 0 ry 90 rz 0 deg; joints [-12.816, -28.462, 112.16, -16.838, -83.104, 51.05]
  Set speed (120.0 mm/s)
  MoveL 11746 to (495.21, 508.59, 20) mm, rotated rx 0 ry 90 rz 0 deg; joints [-12.893, -28.456, 112.123, -16.917, -83.077, 51.068]
  Set speed (15.0 mm/s)
  MoveL 11747 to (496.09, 507.72, 20) mm, rotated rx 0 ry 90 rz 0 deg; joints [-12.795, -28.443, 112.043, -16.821, -83.009, 51.077]
  Set speed (120.0 mm/s)
  MoveL 11748 to (496.2, 508.59, 20) mm, rotated rx 0 ry 90 rz 0 deg; joints [-12.872, -28.437, 112.005, -16.9, -82.981, 51.094]
  Set speed (15.0 mm/s)
  Call Extruder(0.036)
  MoveL 11749 to (497.08, 507.72, 20) mm, rotated rx 0 ry 90 rz 0 deg; joints [-12.774, -28.425, 111.925, -16.804, -82.913, 51.103]
  Set speed (120.0 mm/s)
  MoveL 11750 to (497.19, 508.59, 20) mm, rotated rx 0 ry 90 rz 0 deg; joints [-12.852, -28.419, 111.887, -16.883, -82.886, 51.121]
  Set speed (15.0 mm/s)
  MoveL 11751 to (498.07, 507.72, 20) mm, rotated rx 0 ry 90 rz 0 deg; joints [-12.754, -28.406, 111.807, -16.786, -82.818, 51.13]
  Set speed (120.0 mm/s)
  MoveL 11752 to (498.18, 508.59, 20) mm, rotated rx 0 ry 90 rz 0 deg; joints [-12.831, -28.4, 111.77, -16.865, -82.79, 51.148]
  Set speed (15.0 mm/s)
  MoveL 11753 to (499.06, 507.72, 20) mm, rotated rx 0 ry 90 rz 0 deg; joints [-12.733, -28.387, 111.689, -16.769, -82.722, 51.157]
  Set speed (120.0 mm/s)
  MoveL 11754 to (499.17, 508.59, 20) mm, rotated rx 0 ry 90 rz 0 deg; joints [-12.811, -28.381, 111.651, -16.848, -82.695, 51.175]
  Set speed (15.0 mm/s)
  MoveL 11755 to (500.05, 507.72, 20) mm, rotated rx 0 ry 90 rz 0 deg; joints [-12.713, -28.368, 111.571, -16.753, -82.627, 51.183]
  Set speed (120.0 mm/s)
  MoveL 11756 to (500.16, 508.59, 20) mm, rotated rx 0 ry 90 rz 0 deg; joints [-12.79, -28.362, 111.533, -16.831, -82.599, 51.201]
  Set speed (15.0 mm/s)
  MoveL 11757 to (501.04, 507.72, 20) mm, rotated rx 0 ry 90 rz 0 deg; joints [-12.693, -28.348, 111.453, -16.736, -82.531, 51.21]
  Set speed (120.0 mm/s)
  MoveL 11758 to (501.15, 508.59, 20) mm, rotated rx 0 ry 90 rz 0 deg; joints [-12.77, -28.342, 111.415, -16.815, -82.504, 51.228]
  Set speed (15.0 mm/s)
  MoveL 11759 to (502.03, 507.72, 20) mm, rotated rx 0 ry 90 rz 0 deg; joints [-12.672, -28.329, 111.334, -16.719, -82.436, 51.236]
  Set speed (120.0 mm/s)
  MoveL 11760 to (502.14, 508.59, 20) mm, rotated rx 0 ry 90 rz 0 deg; joints [-12.749, -28.323, 111.297, -16.798, -82.408, 51.254]
  Set speed (15.0 mm/s)
  MoveL 11761 to (503.02, 507.72, 20) mm, rotated rx 0 ry 90 rz 0 deg; joints [-12.652, -28.309, 111.216, -16.703, -82.34, 51.262]
  Set speed (120.0 mm/s)
  MoveL 11762 to (503.13, 508.59, 20) mm, rotated rx 0 ry 90 rz 0 deg; joints [-12.729, -28.303, 111.178, -16.781, -82.313, 51.28]
  Set speed (15.0 mm/s)
  MoveL 11763 to (504.01, 507.72, 20) mm, rotated rx 0 ry 90 rz 0 deg; joints [-12.632, -28.289, 111.097, -16.686, -82.245, 51.288]
  Set speed (120.0 mm/s)
  MoveL 11764 to (504.12, 508.59, 20) mm, rotated rx 0 ry 90 rz 0 deg; joints [-12.709, -28.283, 111.059, -16.765, -82.218, 51.307]
  Set speed (15.0 mm/s)
  MoveL 11765 to (505, 507.72, 20) mm, rotated rx 0 ry 90 rz 0 deg; joints [-12.612, -28.27, 110.978, -16.67, -82.15, 51.315]
  Set speed (120.0 mm/s)
  MoveL 11766 to (505.33, 507.39, 20) mm, rotated rx 0 ry 90 rz 0 deg; joints [-12.575, -28.264, 110.947, -16.633, -82.123, 51.318]
  Set speed (15.0 mm/s)
  Call Extruder(0.134)
  MoveL 11767 to (508.59, 504.12, 20) mm, rotated rx 0 ry 90 rz 0 deg; joints [-12.216, -28.212, 110.641, -16.281, -81.866, 51.345]
  Set speed (120.0 mm/s)
  MoveL 11768 to (508.59, 505.11, 20) mm, rotated rx 0 ry 90 rz 0 deg; joints [-12.305, -28.208, 110.615, -16.372, -81.849, 51.363]
  Set speed (15.0 mm/s)
  Call Extruder(0.143)
  MoveL 11769 to (505.11, 508.59, 20) mm, rotated rx 0 ry 90 rz 0 deg; joints [-12.689, -28.263, 110.941, -16.748, -82.122, 51.333]
  Set speed (120.0 mm/s)
  MoveL 11770 to (506.1, 508.59, 20) mm, rotated rx 0 ry 90 rz 0 deg; joints [-12.668, -28.243, 110.822, -16.732, -82.027, 51.359]
  Set speed (15.0 mm/s)
  Call Extruder(0.103)
  MoveL 11771 to (508.59, 506.1, 20) mm, rotated rx 0 ry 90 rz 0 deg; joints [-12.394, -28.203, 110.589, -16.463, -81.832, 51.38]
  Set speed (120.0 mm/s)
  MoveL 11772 to (508.59, 507.09, 20) mm, rotated rx 0 ry 90 rz 0 deg; joints [-12.483, -28.198, 110.562, -16.554, -81.814, 51.398]
  Set speed (15.0 mm/s)
  Call Extruder(0.062)
  MoveL 11773 to (507.09, 508.59, 20) mm, rotated rx 0 ry 90 rz 0 deg; joints [-12.648, -28.223, 110.703, -16.716, -81.932, 51.385]
  Set speed (120.0 mm/s)
  MoveL 11774 to (508.08, 508.59, 20) mm, rotated rx 0 ry 90 rz 0 deg; joints [-12.628, -28.202, 110.584, -16.7, -81.837, 51.412]
  Set speed (15.0 mm/s)
  Call Extruder(0.021)
  MoveL 11775 to (508.59, 508.08, 20) mm, rotated rx 0 ry 90 rz 0 deg; joints [-12.572, -28.194, 110.536, -16.644, -81.797, 51.416]
  Set speed (120.0 mm/s)
  MoveL 11776 to (505.33, 506.39, 20) mm, rotated rx 0 ry 90 rz 0 deg; joints [-12.485, -28.269, 110.973, -16.542, -82.141, 51.3]
  Set speed (15.0 mm/s)
  Call Extruder(0.134)
  MoveL 11777 to (508.59, 503.13, 20) mm, rotated rx 0 ry 90 rz 0 deg; joints [-12.126, -28.216, 110.666, -16.19, -81.884, 51.328]
  Set speed (120.0 mm/s)
  MoveL 11778 to (508.59, 502.14, 20) mm, rotated rx 0 ry 90 rz 0 deg; joints [-12.037, -28.221, 110.692, -16.099, -81.901, 51.31]
  Set speed (15.0 mm/s)
  Call Extruder(0.136)
  MoveL 11779 to (505.28, 505.46, 20) mm, rotated rx 0 ry 90 rz 0 deg; joints [-12.402, -28.274, 111.004, -16.457, -82.163, 51.283]
  Set speed (120.0 mm/s)
  MoveL 11780 to (504.94, 504.8, 20) mm, rotated rx 0 ry 90 rz 0 deg; joints [-12.349, -28.284, 111.062, -16.402, -82.207, 51.262]
  Set speed (15.0 mm/s)
  Call Extruder(0.150)
  MoveL 11781 to (508.59, 501.15, 20) mm, rotated rx 0 ry 90 rz 0 deg; joints [-11.948, -28.225, 110.717, -16.008, -81.918, 51.293]
  Set speed (120.0 mm/s)
  MoveL 11782 to (508.59, 500.16, 20) mm, rotated rx 0 ry 90 rz 0 deg; joints [-11.858, -28.229, 110.742, -15.917, -81.934, 51.276]
  Set speed (15.0 mm/s)
  Call Extruder(0.164)
  MoveL 11783 to (504.61, 504.15, 20) mm, rotated rx 0 ry 90 rz 0 deg; joints [-12.296, -28.293, 111.119, -16.347, -82.251, 51.242]
  Set speed (120.0 mm/s)
  MoveL 11784 to (504.27, 503.49, 20) mm, rotated rx 0 ry 90 rz 0 deg; joints [-12.243, -28.303, 111.177, -16.292, -82.295, 51.223]
  Set speed (15.0 mm/s)
  Call Extruder(0.178)
  MoveL 11785 to (508.59, 499.17, 20) mm, rotated rx 0 ry 90 rz 0 deg; joints [-11.769, -28.234, 110.767, -15.826, -81.951, 51.259]
  Set speed (120.0 mm/s)
  MoveL 11786 to (508.59, 498.18, 20) mm, rotated rx 0 ry 90 rz 0 deg; joints [-11.679, -28.238, 110.792, -15.735, -81.968, 51.242]
  Set speed (15.0 mm/s)
  Call Extruder(0.192)
  MoveL 11787 to (503.94, 502.84, 20) mm, rotated rx 0 ry 90 rz 0 deg; joints [-12.191, -28.312, 111.234, -16.237, -82.339, 51.203]
  Set speed (120.0 mm/s)
  MoveL 11788 to (503.6, 502.18, 20) mm, rotated rx 0 ry 90 rz 0 deg; joints [-12.138, -28.322, 111.291, -16.181, -82.383, 51.183]
  Set speed (15.0 mm/s)
  Call Extruder(0.205)
  MoveL 11789 to (508.59, 497.19, 20) mm, rotated rx 0 ry 90 rz 0 deg; joints [-11.589, -28.242, 110.817, -15.643, -81.984, 51.225]
  Set speed (120.0 mm/s)
  MoveL 11790 to (508.59, 496.2, 20) mm, rotated rx 0 ry 90 rz 0 deg; joints [-11.5, -28.246, 110.841, -15.552, -82.001, 51.208]
  Set speed (15.0 mm/s)
  Call Extruder(0.219)
  MoveL 11791 to (503.27, 501.53, 20) mm, rotated rx 0 ry 90 rz 0 deg; joints [-12.084, -28.331, 111.348, -16.126, -82.427, 51.163]
  Set speed (120.0 mm/s)
  MoveL 11792 to (502.93, 500.87, 20) mm, rotated rx 0 ry 90 rz 0 deg; joints [-12.031, -28.341, 111.405, -16.071, -82.471, 51.144]
  Set speed (15.0 mm/s)
  Call Extruder(0.233)
  MoveL 11793 to (508.59, 495.21, 20) mm, rotated rx 0 ry 90 rz 0 deg; joints [-11.41, -28.25, 110.865, -15.461, -82.017, 51.192]
  Set speed (120.0 mm/s)
  MoveL 11794 to (508.59, 494.22, 20) mm, rotated rx 0 ry 90 rz 0 deg; joints [-11.32, -28.254, 110.889, -15.369, -82.033, 51.175]
  Set speed (15.0 mm/s)
  Call Extruder(0.247)
  MoveL 11795 to (502.6, 500.22, 20) mm, rotated rx 0 ry 90 rz 0 deg; joints [-11.978, -28.35, 111.462, -16.015, -82.515, 51.124]
  Set speed (120.0 mm/s)
  MoveL 11796 to (502.26, 499.57, 20) mm, rotated rx 0 ry 90 rz 0 deg; joints [-11.925, -28.359, 111.519, -15.96, -82.558, 51.105]
  Set speed (15.0 mm/s)
  Call Extruder(0.109)
  MoveL 11797 to (504.9, 496.92, 20) mm, rotated rx 0 ry 90 rz 0 deg; joints [-11.634, -28.318, 111.268, -15.674, -82.347, 51.128]
  Set speed (120.0 mm/s)
  MoveL 11798 to (505.52, 496.31, 20) mm, rotated rx 0 ry 90 rz 0 deg; joints [-11.567, -28.308, 111.209, -15.608, -82.298, 51.134]
  Set speed (15.0 mm/s)
  Call Extruder(0.127)
  MoveL 11799 to (508.59, 493.23, 20) mm, rotated rx 0 ry 90 rz 0 deg; joints [-11.23, -28.259, 110.913, -15.278, -82.049, 51.159]
  Set speed (120.0 mm/s)
  MoveL 11800 to (508.59, 492.24, 20) mm, rotated rx 0 ry 90 rz 0 deg; joints [-11.14, -28.263, 110.937, -15.186, -82.065, 51.142]
  Set speed (15.0 mm/s)
  MoveL 11801 to (505.52, 495.32, 20) mm, rotated rx 0 ry 90 rz 0 deg; joints [-11.476, -28.312, 111.234, -15.516, -82.315, 51.117]
  Set speed (120.0 mm/s)
  MoveL 11802 to (505.52, 494.33, 20) mm, rotated rx 0 ry 90 rz 0 deg; joints [-11.386, -28.316, 111.258, -15.425, -82.331, 51.101]
  Set speed (15.0 mm/s)
  Call Extruder(0.121)
  MoveL 11803 to (508.44, 491.4, 20) mm, rotated rx 0 ry 90 rz 0 deg; joints [-11.067, -28.269, 110.975, -15.111, -82.093, 51.125]
  Set speed (120.0 mm/s)
  MoveL 11804 to (507.45, 491.4, 20) mm, rotated rx 0 ry 90 rz 0 deg; joints [-11.084, -28.289, 111.094, -15.125, -82.19, 51.101]
  Set speed (15.0 mm/s)
  Call Extruder(0.080)
  MoveL 11805 to (505.52, 493.34, 20) mm, rotated rx 0 ry 90 rz 0 deg; joints [-11.296, -28.32, 111.282, -15.333, -82.347, 51.085]
  Set speed (120.0 mm/s)
  MoveL 11806 to (505.27, 492.6, 20) mm, rotated rx 0 ry 90 rz 0 deg; joints [-11.233, -28.328, 111.33, -15.268, -82.384, 51.067]
  Set speed (15.0 mm/s)
  Call Extruder(0.049)
  MoveL 11807 to (506.46, 491.4, 20) mm, rotated rx 0 ry 90 rz 0 deg; joints [-11.102, -28.309, 111.214, -15.139, -82.286, 51.077]
  Set speed (120.0 mm/s)
  MoveL 11808 to (505.47, 491.4, 20) mm, rotated rx 0 ry 90 rz 0 deg; joints [-11.12, -28.329, 111.333, -15.154, -82.383, 51.053]
  Set speed (15.0 mm/s)
  MoveL 11809 to (504.28, 492.6, 20) mm, rotated rx 0 ry 90 rz 0 deg; joints [-11.251, -28.348, 111.449, -15.283, -82.48, 51.043]
  Set speed (120.0 mm/s)
  MoveL 11810 to (503.29, 492.6, 20) mm, rotated rx 0 ry 90 rz 0 deg; joints [-11.269, -28.367, 111.568, -15.297, -82.577, 51.018]
  Set speed (15.0 mm/s)
  MoveL 11811 to (504.48, 491.4, 20) mm, rotated rx 0 ry 90 rz 0 deg; joints [-11.137, -28.348, 111.452, -15.168, -82.479, 51.029]
  Set speed (120.0 mm/s)
  MoveL 11812 to (503.49, 491.4, 20) mm, rotated rx 0 ry 90 rz 0 deg; joints [-11.155, -28.368, 111.571, -15.183, -82.576, 51.004]
  Set speed (15.0 mm/s)
  MoveL 11813 to (502.3, 492.6, 20) mm, rotated rx 0 ry 90 rz 0 deg; joints [-11.287, -28.386, 111.686, -15.312, -82.673, 50.994]
  Set speed (120.0 mm/s)
  MoveL 11814 to (501.31, 492.6, 20) mm, rotated rx 0 ry 90 rz 0 deg; joints [-11.305, -28.405, 111.805, -15.327, -82.77, 50.969]
  Set speed (15.0 mm/s)
  MoveL 11815 to (502.5, 491.4, 20) mm, rotated rx 0 ry 90 rz 0 deg; joints [-11.173, -28.387, 111.69, -15.198, -82.673, 50.98]
  Set speed (120.0 mm/s)
  MoveL 11816 to (501.51, 491.4, 20) mm, rotated rx 0 ry 90 rz 0 deg; joints [-11.191, -28.406, 111.809, -15.212, -82.769, 50.956]
  Set speed (15.0 mm/s)
  MoveL 11817 to (500.32, 492.6, 20) mm, rotated rx 0 ry 90 rz 0 deg; joints [-11.323, -28.424, 111.924, -15.342, -82.867, 50.945]
  Set speed (120.0 mm/s)
  MoveL 11818 to (499.33, 492.6, 20) mm, rotated rx 0 ry 90 rz 0 deg; joints [-11.342, -28.443, 112.042, -15.357, -82.963, 50.92]
  Set speed (15.0 mm/s)
  MoveL 11819 to (500.52, 491.4, 20) mm, rotated rx 0 ry 90 rz 0 deg; joints [-11.209, -28.425, 111.927, -15.227, -82.866, 50.931]
  Set speed (120.0 mm/s)
  MoveL 11820 to (499.53, 491.4, 20) mm, rotated rx 0 ry 90 rz 0 deg; joints [-11.227, -28.444, 112.046, -15.242, -82.963, 50.907]
  Set speed (15.0 mm/s)
  Call Extruder(0.049)
  MoveL 11821 to (498.34, 492.6, 20) mm, rotated rx 0 ry 90 rz 0 deg; joints [-11.36, -28.462, 112.16, -15.372, -83.06, 50.896]
  Set speed (120.0 mm/s)
  MoveL 11822 to (497.35, 492.6, 20) mm, rotated rx 0 ry 90 rz 0 deg; joints [-11.378, -28.48, 112.278, -15.388, -83.157, 50.871]
  Set speed (15.0 mm/s)
  MoveL 11823 to (498.54, 491.4, 20) mm, rotated rx 0 ry 90 rz 0 deg; joints [-11.245, -28.462, 112.164, -15.257, -83.06, 50.882]
  Set speed (120.0 mm/s)
  MoveL 11824 to (497.55, 491.4, 20) mm, rotated rx 0 ry 90 rz 0 deg; joints [-11.264, -28.481, 112.282, -15.272, -83.156, 50.858]
  Set speed (15.0 mm/s)
  MoveL 11825 to (496.36, 492.6, 20) mm, rotated rx 0 ry 90 rz 0 deg; joints [-11.397, -28.498, 112.396, -15.403, -83.253, 50.846]
  MoveL 11826 to (496.23, 492.73, 20) mm, rotated rx 0 ry 90 rz 0 deg; joints [-11.41, -28.5, 112.408, -15.417, -83.263, 50.845]
  Set speed (120.0 mm/s)
  MoveL 11827 to (504.54, 493.58, 20) mm, rotated rx 0 ry 90 rz 0 deg; joints [-11.335, -28.339, 111.393, -15.369, -82.438, 51.065]
  Set speed (1000.0 mm/s)
  MoveL 11828 to (504.54, 495.95, 20) mm, rotated rx 0 ry 90 rz 0 deg; joints [-11.552, -28.329, 111.336, -15.589, -82.399, 51.103]
  Set speed (1000.0 mm/s)
  MoveL 11829 to (501.26, 497.6, 20) mm, rotated rx 0 ry 90 rz 0 deg; joints [-11.764, -28.387, 111.689, -15.793, -82.69, 51.047]
  Set speed (15.0 mm/s)
  Call Extruder(0.028)
  MoveL 11830 to (501.93, 496.92, 20) mm, rotated rx 0 ry 90 rz 0 deg; joints [-11.69, -28.376, 111.624, -15.72, -82.636, 51.054]
  Set speed (120.0 mm/s)
  MoveL 11831 to (502.92, 496.92, 20) mm, rotated rx 0 ry 90 rz 0 deg; joints [-11.671, -28.357, 111.506, -15.705, -82.54, 51.079]
  Set speed (15.0 mm/s)
  Call Extruder(0.055)
  MoveL 11832 to (501.59, 498.26, 20) mm, rotated rx 0 ry 90 rz 0 deg; joints [-11.818, -28.378, 111.632, -15.849, -82.646, 51.066]
  Set speed (120.0 mm/s)
  MoveL 11833 to (501.93, 498.91, 20) mm, rotated rx 0 ry 90 rz 0 deg; joints [-11.871, -28.368, 111.576, -15.904, -82.602, 51.086]
  Set speed (15.0 mm/s)
  Call Extruder(0.082)
  MoveL 11834 to (503.91, 496.92, 20) mm, rotated rx 0 ry 90 rz 0 deg; joints [-11.652, -28.338, 111.387, -15.689, -82.444, 51.104]
  MoveL 11835 to (504.04, 496.8, 20) mm, rotated rx 0 ry 90 rz 0 deg; joints [-11.639, -28.336, 111.375, -15.676, -82.434, 51.105]
  Set speed (30.0 mm/s)
  Call Extruder(-0.400)
  MoveL 11836 to (504.04, 496.8, 20) mm, rotated rx 0 ry 90 rz 0 deg; joints [-11.639, -28.336, 111.375, -15.676, -82.434, 51.105]
  Call M_RunCode(82)
  Call M_RunCode(107)
  Call M_RunCode(104)
  Call SetRPM(0.0)
  Call M_RunCode(140)
  Call SetRPM(0.0)
  Call Extruder(1.000)
  Call Extruder(-0.500)
  Set speed (5.0 mm/s)
  MoveL 11837 to (504.04, 496.8, 20) mm, rotated rx 0 ry 90 rz 0 deg; joints [-11.639, -28.336, 111.375, -15.676, -82.434, 51.105]
  Set speed (1000.0 mm/s)
  MoveL 11838 to (504.04, 496.8, 20) mm, rotated rx 0 ry 90 rz 0 deg; joints [-11.639, -28.336, 111.375, -15.676, -82.434, 51.105]
  Call M_RunCode(82)
  Call M_RunCode(104)
  Call SetRPM(0.0)
